C05458=1043.146,323.202,382.853,172.338,41.617,158.001
C05459=1043.153,323.449,382.817,172.342,41.620,158.002
C05460=1043.160,323.697,382.782,172.346,41.623,158.003
C05461=1043.167,323.944,382.748,172.350,41.626,158.003
C05462=1043.174,324.192,382.713,172.355,41.629,158.004
C05463=1043.181,324.439,382.679,172.359,41.631,158.005
C05464=1043.189,324.687,382.643,172.364,41.634,158.006
C05465=1043.196,324.934,382.609,172.369,41.637,158.007
C05466=1043.203,325.181,382.574,172.373,41.640,158.008
C05467=1043.210,325.429,382.538,172.377,41.643,158.009
C05468=1043.218,325.677,382.504,172.382,41.645,158.010
C05469=1043.225,325.924,382.468,172.386,41.649,158.011
C05470=1043.232,326.171,382.434,172.390,41.652,158.012
C05471=1043.239,326.419,382.399,172.395,41.654,158.013
C05472=1043.247,326.667,382.365,172.399,41.657,158.014
C05473=1043.254,326.914,382.329,172.403,41.660,158.014
C05474=1043.260,327.161,382.294,172.408,41.663,158.015
C05475=1043.268,327.408,382.260,172.412,41.666,158.016
C05476=1043.275,327.656,382.224,172.416,41.669,158.017
C05477=1043.283,327.903,382.189,172.422,41.672,158.018
C05478=1043.290,328.150,382.154,172.425,41.675,158.019
C05479=1043.297,328.398,382.118,172.431,41.678,158.020
C05480=1043.305,328.645,382.084,172.435,41.681,158.021
C05481=1043.312,328.894,382.048,172.439,41.683,158.022
C05482=1043.319,329.141,382.013,172.444,41.686,158.023
C05483=1043.326,329.388,381.978,172.448,41.689,158.024
C05484=1043.334,329.635,381.942,172.452,41.693,158.025
C05485=1043.341,329.883,381.907,172.457,41.696,158.026
C05486=1043.348,330.130,381.872,172.461,41.699,158.027
C05487=1043.355,330.378,381.836,172.467,41.702,158.028
C05488=1043.362,330.625,381.801,172.471,41.705,158.029
C05489=1043.369,330.872,381.766,172.475,41.708,158.030
C05490=1043.376,331.120,381.729,172.480,41.711,158.031
C05491=1043.382,331.367,381.694,172.484,41.714,158.032
C05492=1043.389,331.614,381.658,172.489,41.717,158.033
C05493=1043.397,331.862,381.622,172.493,41.720,158.034
C05494=1043.404,332.109,381.587,172.498,41.723,158.035
C05495=1043.411,332.357,381.551,172.503,41.726,158.036
C05496=1043.418,332.604,381.515,172.507,41.730,158.037
C05497=1043.425,332.851,381.480,172.512,41.733,158.038
C05498=1043.433,333.099,381.444,172.516,41.736,158.039
C05499=1043.443,333.428,381.396,172.523,41.740,158.040
C05500=1043.452,333.760,381.349,172.528,41.744,158.041
C05501=1043.462,334.090,381.301,172.535,41.749,158.043
C05502=1043.472,334.420,381.253,172.541,41.753,158.044
C05503=1043.479,334.667,381.217,172.546,41.756,158.045
C05504=1043.486,334.915,381.182,172.551,41.759,158.046
C05505=1043.493,335.162,381.146,172.555,41.762,158.047
C05506=1043.501,335.409,381.110,172.560,41.765,158.048
C05507=1043.508,335.656,381.074,172.564,41.768,158.049
C05508=1043.515,335.904,381.038,172.569,41.772,158.050
C05509=1043.522,336.151,381.002,172.574,41.775,158.051
C05510=1043.529,336.399,380.966,172.578,41.778,158.052
C05511=1043.536,336.645,380.930,172.583,41.782,158.053
C05512=1043.543,336.893,380.893,172.588,41.785,158.054
C05513=1043.550,337.140,380.857,172.593,41.788,158.055
C05514=1043.558,337.387,380.821,172.598,41.792,158.057
C05515=1043.565,337.635,380.784,172.602,41.795,158.058
C05516=1043.572,337.882,380.748,172.608,41.798,158.059
C05517=1043.580,338.129,380.712,172.612,41.801,158.060
C05518=1043.588,338.377,380.676,172.617,41.804,158.061
C05519=1043.594,338.624,380.639,172.621,41.808,158.062
C05520=1043.602,338.871,380.603,172.626,41.811,158.063
C05521=1043.609,339.118,380.567,172.631,41.815,158.064
C05522=1043.616,339.366,380.531,172.636,41.818,158.065
C05523=1043.623,339.613,380.494,172.640,41.821,158.066
C05524=1043.631,339.861,380.458,172.645,41.824,158.067
C05525=1043.637,340.108,380.422,172.651,41.828,158.068
C05526=1043.645,340.355,380.385,172.655,41.831,158.069
C05527=1043.653,340.602,380.349,172.660,41.835,158.070
C05528=1043.660,340.849,380.313,172.665,41.838,158.072
C05529=1043.667,341.096,380.276,172.670,41.841,158.073
C05530=1043.675,341.344,380.240,172.675,41.845,158.074
C05531=1043.682,341.591,380.203,172.679,41.848,158.075
C05532=1043.689,341.838,380.166,172.685,41.851,158.076
C05533=1043.697,342.085,380.130,172.689,41.855,158.077
C05534=1043.704,342.333,380.093,172.694,41.858,158.078
C05535=1043.711,342.580,380.056,172.699,41.862,158.079
C05536=1043.718,342.828,380.020,172.704,41.865,158.080
C05537=1043.726,343.074,379.983,172.709,41.869,158.081
C05538=1043.733,343.321,379.946,172.714,41.872,158.082
C05539=1043.741,343.568,379.909,172.719,41.875,158.084
C05540=1043.748,343.816,379.872,172.724,41.879,158.085
C05541=1043.755,344.063,379.835,172.729,41.883,158.086
C05542=1043.762,344.310,379.799,172.734,41.886,158.087
C05543=1043.769,344.557,379.761,172.739,41.889,158.088
C05544=1043.777,344.804,379.725,172.744,41.893,158.089
C05545=1043.784,345.052,379.688,172.749,41.896,158.090
C05546=1043.792,345.299,379.652,172.754,41.900,158.092
C05547=1043.799,345.546,379.614,172.759,41.904,158.093
C05548=1043.806,345.793,379.576,172.764,41.907,158.094
C05549=1043.814,346.041,379.540,172.769,41.911,158.095
C05550=1043.821,346.288,379.503,172.775,41.914,158.096
C05551=1043.828,346.534,379.466,172.779,41.918,158.097
C05552=1043.836,346.781,379.429,172.784,41.921,158.099
C05553=1043.843,347.029,379.392,172.790,41.925,158.100
C05554=1043.850,347.276,379.354,172.795,41.929,158.101
C05555=1043.860,347.603,379.305,172.802,41.933,158.102
C05556=1043.870,347.929,379.256,172.809,41.938,158.104
C05557=1043.880,348.256,379.207,172.815,41.943,158.106
C05558=1043.890,348.583,379.158,172.821,41.947,158.107
C05559=1043.897,348.830,379.120,172.827,41.952,158.108
C05560=1043.905,349.077,379.083,172.832,41.955,158.109
C05561=1043.912,349.324,379.046,172.838,41.959,158.111
C05562=1043.920,349.571,379.008,172.843,41.962,158.112
C05563=1043.927,349.818,378.971,172.847,41.966,158.113
C05564=1043.935,350.065,378.934,172.853,41.969,158.114
C05565=1043.942,350.312,378.896,172.858,41.973,158.115
C05566=1043.949,350.559,378.859,172.864,41.977,158.117
C05567=1043.957,350.807,378.821,172.869,41.980,158.118
C05568=1043.965,351.054,378.783,172.874,41.985,158.119
C05569=1043.972,351.301,378.745,172.879,41.988,158.120
C05570=1043.979,351.548,378.708,172.884,41.992,158.121
C05571=1043.987,351.795,378.671,172.890,41.996,158.123
C05572=1043.994,352.042,378.633,172.895,41.999,158.124
C05573=1044.002,352.288,378.595,172.901,42.003,158.125
C05574=1044.009,352.535,378.557,172.905,42.007,158.126
C05575=1044.017,352.783,378.519,172.911,42.011,158.128
C05576=1044.025,353.030,378.481,172.916,42.015,158.129
C05577=1044.032,353.277,378.444,172.922,42.019,158.130
C05578=1044.039,353.523,378.405,172.927,42.022,158.131
C05579=1044.047,353.771,378.368,172.933,42.026,158.133
C05580=1044.055,354.018,378.330,172.938,42.030,158.134
C05581=1044.062,354.265,378.292,172.944,42.034,158.135
C05582=1044.069,354.512,378.254,172.948,42.038,158.136
C05583=1044.077,354.759,378.216,172.954,42.042,158.138
C05584=1044.085,355.006,378.178,172.959,42.046,158.139
C05585=1044.092,355.253,378.140,172.965,42.049,158.140
C05586=1044.100,355.500,378.102,172.970,42.053,158.142
C05587=1044.107,355.747,378.064,172.976,42.057,158.143
C05588=1044.115,355.994,378.025,172.981,42.061,158.144
C05589=1044.122,356.241,377.988,172.987,42.065,158.145
C05590=1044.131,356.487,377.950,172.992,42.069,158.147
C05591=1044.139,356.734,377.912,172.998,42.073,158.148
C05592=1044.145,356.982,377.874,173.003,42.077,158.149
C05593=1044.153,357.228,377.835,173.009,42.081,158.151
C05594=1044.161,357.475,377.797,173.015,42.085,158.152
C05595=1044.169,357.722,377.758,173.020,42.089,158.153
C05596=1044.177,357.970,377.721,173.026,42.093,158.155
C05597=1044.184,358.216,377.682,173.031,42.096,158.156
C05598=1044.192,358.463,377.644,173.037,42.100,158.157
C05599=1044.199,358.710,377.605,173.042,42.105,158.158
C05600=1044.207,358.957,377.567,173.048,42.109,158.160
C05601=1044.215,359.204,377.528,173.054,42.113,158.161
C05602=1044.222,359.451,377.490,173.059,42.117,158.162
C05603=1044.230,359.698,377.451,173.065,42.121,158.164
C05604=1044.238,359.944,377.413,173.070,42.125,158.165
C05605=1044.245,360.191,377.374,173.076,42.129,158.166
C05606=1044.253,360.438,377.335,173.082,42.133,158.168
C05607=1044.261,360.685,377.297,173.087,42.138,158.169
C05608=1044.269,360.932,377.259,173.093,42.142,158.171
C05609=1044.276,361.180,377.219,173.099,42.146,158.172
C05610=1044.284,361.426,377.180,173.104,42.150,158.173
C05611=1044.294,361.758,377.129,173.112,42.155,158.175
C05612=1044.305,362.091,377.077,173.120,42.161,158.177
C05613=1044.315,362.423,377.024,173.128,42.166,158.179
C05614=1044.326,362.755,376.972,173.135,42.172,158.181
C05615=1044.333,363.003,376.932,173.141,42.177,158.182
C05616=1044.341,363.249,376.894,173.147,42.181,158.184
C05617=1044.349,363.496,376.854,173.153,42.185,158.185
C05618=1044.356,363.743,376.816,173.159,42.189,158.186
C05619=1044.365,363.989,376.777,173.165,42.193,158.188
C05620=1044.372,364.237,376.738,173.170,42.198,158.189
C05621=1044.380,364.483,376.699,173.176,42.202,158.191
C05622=1044.387,364.730,376.659,173.182,42.206,158.192
C05623=1044.396,364.977,376.620,173.187,42.211,158.193
C05624=1044.403,365.223,376.580,173.194,42.215,158.195
C05625=1044.411,365.470,376.542,173.200,42.219,158.196
C05626=1044.419,365.717,376.502,173.206,42.224,158.198
C05627=1044.425,365.964,376.463,173.212,42.228,158.199
C05628=1044.434,366.210,376.424,173.217,42.232,158.201
C05629=1044.442,366.457,376.384,173.223,42.237,158.202
C05630=1044.450,366.703,376.345,173.230,42.241,158.204
C05631=1044.457,366.951,376.306,173.235,42.245,158.205
C05632=1044.465,367.197,376.266,173.241,42.250,158.207
C05633=1044.473,367.444,376.226,173.247,42.255,158.208
C05634=1044.482,367.691,376.187,173.254,42.258,158.209
C05635=1044.489,367.937,376.148,173.260,42.263,158.211
C05636=1044.497,368.184,376.108,173.265,42.268,158.212
C05637=1044.505,368.431,376.069,173.271,42.272,158.214
C05638=1044.513,368.678,376.030,173.278,42.277,158.215
C05639=1044.521,368.925,375.990,173.284,42.281,158.217
C05640=1044.529,369.171,375.950,173.289,42.285,158.218
C05641=1044.537,369.418,375.911,173.296,42.290,158.220
C05642=1044.545,369.665,375.871,173.302,42.294,158.221
C05643=1044.552,369.911,375.832,173.308,42.299,158.223
C05644=1044.560,370.158,375.792,173.314,42.303,158.224
C05645=1044.569,370.404,375.752,173.321,42.308,158.226
C05646=1044.577,370.651,375.712,173.327,42.312,158.227
C05647=1044.585,370.897,375.672,173.333,42.317,158.229
C05648=1044.593,371.144,375.633,173.339,42.321,158.230
C05649=1044.601,371.391,375.593,173.345,42.327,158.232
C05650=1044.609,371.637,375.552,173.352,42.331,158.234
C05651=1044.616,371.884,375.512,173.358,42.336,158.235
C05652=1044.624,372.131,375.472,173.364,42.340,158.237
C05653=1044.633,372.377,375.432,173.371,42.345,158.238
C05654=1044.641,372.624,375.392,173.377,42.350,158.240
C05655=1044.649,372.870,375.352,173.383,42.354,158.241
C05656=1044.656,373.117,375.312,173.389,42.359,158.243
C05657=1044.664,373.364,375.271,173.395,42.364,158.245
C05658=1044.672,373.611,375.231,173.402,42.368,158.246
C05659=1044.680,373.857,375.190,173.408,42.373,158.248
C05660=1044.688,374.104,375.151,173.414,42.378,158.249
C05661=1044.697,374.350,375.111,173.421,42.383,158.251
C05662=1044.705,374.597,375.070,173.427,42.388,158.253
C05663=1044.713,374.844,375.030,173.434,42.393,158.254
C05664=1044.721,375.090,374.989,173.440,42.397,158.256
C05665=1044.729,375.336,374.948,173.447,42.402,158.258
C05666=1044.737,375.583,374.908,173.453,42.407,158.259
C05667=1044.748,375.935,374.850,173.462,42.414,158.261
C05668=1044.760,376.287,374.793,173.472,42.421,158.264
C05669=1044.772,376.639,374.734,173.481,42.427,158.266
C05670=1044.783,376.991,374.676,173.490,42.434,158.268
C05671=1044.792,377.237,374.636,173.497,42.439,158.270
C05672=1044.800,377.483,374.596,173.504,42.444,158.272
C05673=1044.809,377.730,374.555,173.510,42.449,158.273
C05674=1044.817,377.976,374.514,173.517,42.454,158.275
C05675=1044.825,378.223,374.473,173.524,42.459,158.277
C05676=1044.833,378.470,374.432,173.530,42.464,158.278
C05677=1044.841,378.716,374.392,173.537,42.469,158.280
C05678=1044.849,378.962,374.351,173.543,42.474,158.282
C05679=1044.858,379.209,374.310,173.550,42.479,158.283
C05680=1044.866,379.455,374.270,173.557,42.484,158.285
C05681=1044.874,379.702,374.229,173.563,42.489,158.287
C05682=1044.882,379.948,374.187,173.570,42.494,158.289
C05683=1044.890,380.195,374.146,173.576,42.499,158.290
C05684=1044.898,380.441,374.105,173.584,42.504,158.292
C05685=1044.907,380.687,374.064,173.591,42.509,158.294
C05686=1044.915,380.934,374.022,173.597,42.514,158.296
C05687=1044.924,381.180,373.981,173.604,42.519,158.297
C05688=1044.932,381.427,373.940,173.610,42.525,158.299
C05689=1044.940,381.674,373.899,173.617,42.530,158.301
C05690=1044.948,381.920,373.857,173.624,42.535,158.303
C05691=1044.956,382.165,373.816,173.632,42.540,158.304
C05692=1044.965,382.412,373.775,173.638,42.545,158.306
C05693=1044.973,382.658,373.733,173.645,42.550,158.308
C05694=1044.981,382.905,373.692,173.652,42.556,158.310
C05695=1044.990,383.151,373.650,173.658,42.561,158.311
C05696=1044.998,383.397,373.609,173.666,42.566,158.313
C05697=1045.006,383.644,373.567,173.673,42.571,158.315
C05698=1045.014,383.890,373.526,173.680,42.577,158.317
C05699=1045.023,384.136,373.484,173.686,42.582,158.319
C05700=1045.032,384.382,373.443,173.694,42.587,158.320
C05701=1045.040,384.629,373.401,173.701,42.593,158.322
C05702=1045.049,384.876,373.359,173.708,42.598,158.324
C05703=1045.057,385.121,373.318,173.714,42.603,158.326
C05704=1045.065,385.368,373.276,173.722,42.609,158.328
C05705=1045.074,385.615,373.234,173.729,42.614,158.330
C05706=1045.082,385.860,373.193,173.736,42.620,158.332
C05707=1045.091,386.107,373.151,173.743,42.625,158.333
C05708=1045.099,386.353,373.109,173.751,42.630,158.335
C05709=1045.108,386.600,373.067,173.757,42.636,158.337
C05710=1045.117,386.845,373.026,173.764,42.641,158.339
C05711=1045.125,387.092,372.983,173.772,42.647,158.341
C05712=1045.134,387.338,372.942,173.779,42.652,158.343
C05713=1045.143,387.585,372.900,173.786,42.658,158.345
C05714=1045.151,387.831,372.857,173.794,42.663,158.347
C05715=1045.160,388.077,372.815,173.801,42.669,158.348
C05716=1045.169,388.323,372.774,173.808,42.674,158.350
C05717=1045.177,388.569,372.731,173.816,42.679,158.352
C05718=1045.186,388.815,372.689,173.823,42.685,158.354
C05719=1045.194,389.062,372.647,173.831,42.691,158.356
C05720=1045.203,389.308,372.605,173.838,42.696,158.358
C05721=1045.212,389.554,372.562,173.844,42.702,158.360
C05722=1045.220,389.801,372.520,173.852,42.708,158.362
C05723=1045.231,390.093,372.469,173.861,42.714,158.364
C05724=1045.241,390.386,372.419,173.870,42.721,158.367
C05725=1045.251,390.679,372.368,173.879,42.728,158.369
C05726=1045.261,390.971,372.318,173.888,42.735,158.371
C05727=1045.270,391.218,372.275,173.895,42.740,158.373
C05728=1045.279,391.464,372.233,173.903,42.746,158.375
C05729=1045.287,391.710,372.190,173.910,42.752,158.377
C05730=1045.296,391.956,372.147,173.917,42.758,158.379
C05731=1045.305,392.202,372.105,173.925,42.763,158.381
C05732=1045.313,392.448,372.062,173.934,42.769,158.383
C05733=1045.322,392.694,372.019,173.941,42.775,158.385
C05734=1045.331,392.941,371.976,173.949,42.781,158.387
C05735=1045.340,393.187,371.933,173.956,42.787,158.389
C05736=1045.349,393.433,371.890,173.964,42.793,158.391
C05737=1045.357,393.679,371.847,173.971,42.799,158.394
C05738=1045.366,393.925,371.804,173.979,42.805,158.396
C05739=1045.375,394.171,371.762,173.987,42.811,158.398
C05740=1045.383,394.417,371.719,173.994,42.817,158.400
C05741=1045.392,394.663,371.675,174.003,42.822,158.402
C05742=1045.401,394.910,371.632,174.010,42.828,158.404
C05743=1045.411,395.155,371.589,174.018,42.834,158.406
C05744=1045.419,395.401,371.546,174.026,42.840,158.408
C05745=1045.428,395.647,371.503,174.033,42.846,158.410
C05746=1045.437,395.893,371.460,174.042,42.852,158.412
C05747=1045.445,396.139,371.416,174.050,42.858,158.414
C05748=1045.454,396.385,371.373,174.057,42.864,158.417
C05749=1045.463,396.631,371.329,174.065,42.871,158.419
C05750=1045.472,396.877,371.286,174.074,42.877,158.421
C05751=1045.481,397.123,371.242,174.081,42.883,158.423
C05752=1045.490,397.369,371.199,174.089,42.889,158.425
C05753=1045.499,397.615,371.155,174.097,42.895,158.427
C05754=1045.508,397.862,371.111,174.106,42.901,158.430
C05755=1045.516,398.107,371.068,174.114,42.908,158.432
C05756=1045.526,398.352,371.025,174.121,42.914,158.434
C05757=1045.535,398.599,370.981,174.130,42.920,158.436
C05758=1045.544,398.844,370.937,174.138,42.926,158.438
C05759=1045.553,399.090,370.893,174.145,42.932,158.440
C05760=1045.562,399.336,370.850,174.154,42.939,158.443
C05761=1045.571,399.583,370.806,174.162,42.945,158.445
C05762=1045.580,399.828,370.762,174.171,42.952,158.447
C05763=1045.589,400.074,370.718,174.179,42.957,158.449
C05764=1045.599,400.320,370.674,174.187,42.964,158.452
C05765=1045.608,400.566,370.630,174.195,42.970,158.454
C05766=1045.616,400.812,370.586,174.203,42.977,158.456
C05767=1045.625,401.058,370.542,174.212,42.983,158.458
C05768=1045.635,401.304,370.498,174.220,42.989,158.461
C05769=1045.644,401.550,370.454,174.229,42.996,158.463
C05770=1045.653,401.795,370.410,174.237,43.003,158.465
C05771=1045.662,402.041,370.366,174.246,43.009,158.468
C05772=1045.671,402.287,370.321,174.254,43.015,158.470
C05773=1045.681,402.533,370.276,174.263,43.022,158.472
C05774=1045.689,402.779,370.233,174.271,43.029,158.475
C05775=1045.702,403.117,370.171,174.283,43.037,158.478
C05776=1045.715,403.456,370.110,174.294,43.047,158.481
C05777=1045.728,403.793,370.049,174.306,43.056,158.484
C05778=1045.740,404.131,369.988,174.318,43.065,158.488
C05779=1045.756,404.536,369.914,174.332,43.076,158.492
C05780=1045.770,404.941,369.840,174.346,43.087,158.496
C05781=1045.786,405.345,369.767,174.360,43.098,158.500
C05782=1045.802,405.749,369.693,174.376,43.109,158.504
C05783=1045.810,405.995,369.647,174.384,43.116,158.506
C05784=1045.820,406.241,369.603,174.393,43.123,158.508
C05785=1045.829,406.487,369.558,174.402,43.130,158.511
C05786=1045.839,406.732,369.513,174.410,43.137,158.513
C05787=1045.848,406.978,369.468,174.419,43.144,158.516
C05788=1045.857,407.223,369.423,174.428,43.150,158.518
C05789=1045.866,407.469,369.377,174.438,43.157,158.521
C05790=1045.876,407.715,369.333,174.447,43.164,158.523
C05791=1045.885,407.961,369.287,174.455,43.172,158.526
C05792=1045.895,408.206,369.242,174.464,43.178,158.528
C05793=1045.904,408.452,369.198,174.473,43.185,158.531
C05794=1045.914,408.697,369.151,174.483,43.192,158.533
C05795=1045.924,408.943,369.106,174.492,43.199,158.536
C05796=1045.933,409.189,369.061,174.500,43.207,158.539
C05797=1045.943,409.434,369.016,174.509,43.213,158.541
C05798=1045.952,409.680,368.970,174.519,43.221,158.544
C05799=1045.962,409.926,368.925,174.528,43.228,158.546
C05800=1045.971,410.172,368.879,174.537,43.235,158.549
C05801=1045.981,410.417,368.834,174.547,43.242,158.552
C05802=1045.991,410.663,368.788,174.556,43.249,158.554
C05803=1046.001,410.908,368.742,174.565,43.256,158.557
C05804=1046.010,411.155,368.697,174.575,43.263,158.559
C05805=1046.020,411.400,368.650,174.584,43.271,158.562
C05806=1046.030,411.645,368.605,174.594,43.278,158.565
C05807=1046.039,411.891,368.559,174.603,43.285,158.567
C05808=1046.050,412.137,368.513,174.613,43.292,158.570
C05809=1046.059,412.383,368.468,174.622,43.300,158.573
C05810=1046.070,412.628,368.422,174.631,43.307,158.575
C05811=1046.079,412.873,368.376,174.641,43.315,158.578
C05812=1046.089,413.119,368.329,174.650,43.322,158.581
C05813=1046.098,413.364,368.283,174.661,43.329,158.583
C05814=1046.108,413.610,368.237,174.671,43.337,158.586
C05815=1046.117,413.856,368.190,174.680,43.344,158.589
C05816=1046.128,414.101,368.145,174.690,43.352,158.592
C05817=1046.137,414.346,368.098,174.699,43.359,158.594
C05818=1046.147,414.592,368.052,174.709,43.367,158.597
C05819=1046.157,414.838,368.005,174.719,43.375,158.600
C05820=1046.166,415.083,367.959,174.729,43.382,158.603
C05821=1046.176,415.329,367.912,174.739,43.389,158.606
C05822=1046.186,415.575,367.866,174.748,43.397,158.608
C05823=1046.197,415.819,367.819,174.758,43.405,158.611
C05824=1046.206,416.065,367.773,174.769,43.412,158.614
C05825=1046.217,416.310,367.726,174.778,43.420,158.617
C05826=1046.227,416.556,367.679,174.788,43.428,158.620
C05827=1046.236,416.801,367.632,174.799,43.436,158.623
C05828=1046.246,417.046,367.586,174.809,43.443,158.626
C05829=1046.256,417.292,367.539,174.818,43.451,158.628
C05830=1046.266,417.538,367.492,174.829,43.459,158.631
C05831=1046.277,417.783,367.445,174.839,43.466,158.634
C05832=1046.287,418.028,367.398,174.850,43.474,158.637
C05833=1046.297,418.274,367.352,174.859,43.482,158.640
C05834=1046.307,418.519,367.305,174.870,43.490,158.643
C05835=1046.324,418.930,367.225,174.888,43.503,158.648
C05836=1046.341,419.343,367.145,174.904,43.517,158.653
C05837=1046.358,419.754,367.066,174.922,43.530,158.658
C05838=1046.375,420.166,366.986,174.940,43.544,158.663
C05839=1046.386,420.412,366.939,174.951,43.552,158.666
C05840=1046.396,420.657,366.892,174.962,43.560,158.669
C05841=1046.405,420.902,366.844,174.972,43.568,158.672
C05842=1046.416,421.147,366.796,174.983,43.576,158.676
C05843=1046.426,421.392,366.749,174.994,43.584,158.679
C05844=1046.436,421.638,366.702,175.004,43.593,158.682
C05845=1046.447,421.883,366.653,175.015,43.601,158.685
C05846=1046.457,422.128,366.606,175.026,43.609,158.688
C05847=1046.467,422.373,366.558,175.036,43.617,158.691
C05848=1046.477,422.619,366.510,175.047,43.625,158.694
C05849=1046.489,422.864,366.462,175.058,43.634,158.697
C05850=1046.499,423.109,366.414,175.069,43.642,158.700
C05851=1046.509,423.354,366.367,175.080,43.651,158.704
C05852=1046.520,423.599,366.319,175.090,43.659,158.707
C05853=1046.530,423.844,366.270,175.102,43.667,158.710
C05854=1046.541,424.090,366.222,175.113,43.676,158.713
C05855=1046.552,424.334,366.174,175.124,43.684,158.717
C05856=1046.562,424.580,366.126,175.135,43.693,158.720
C05857=1046.572,424.825,366.078,175.147,43.701,158.723
C05858=1046.583,425.071,366.030,175.158,43.710,158.726
C05859=1046.594,425.315,365.981,175.169,43.718,158.730
C05860=1046.604,425.560,365.932,175.181,43.727,158.733
C05861=1046.615,425.805,365.884,175.192,43.735,158.736
C05862=1046.625,426.051,365.835,175.203,43.744,158.739
C05863=1046.636,426.296,365.787,175.215,43.753,158.743
C05864=1046.647,426.540,365.738,175.226,43.761,158.746
C05865=1046.658,426.786,365.689,175.238,43.770,158.750
C05866=1046.668,427.030,365.641,175.249,43.779,158.753
C05867=1046.679,427.275,365.592,175.261,43.788,158.756
C05868=1046.690,427.520,365.543,175.273,43.797,158.760
C05869=1046.701,427.766,365.494,175.284,43.805,158.763
C05870=1046.711,428.010,365.445,175.296,43.814,158.767
C05871=1046.723,428.255,365.396,175.308,43.823,158.770
C05872=1046.733,428.500,365.347,175.319,43.832,158.773
C05873=1046.744,428.745,365.298,175.332,43.841,158.777
C05874=1046.755,428.990,365.249,175.343,43.850,158.780
C05875=1046.766,429.235,365.199,175.355,43.859,158.784
C05876=1046.777,429.479,365.150,175.368,43.868,158.787
C05877=1046.787,429.724,365.101,175.379,43.877,158.791
C05878=1046.798,429.969,365.051,175.391,43.886,158.794
C05879=1046.809,430.214,365.002,175.404,43.895,158.798
C05880=1046.820,430.459,364.953,175.416,43.904,158.802
C05881=1046.831,430.704,364.903,175.427,43.914,158.805
C05882=1046.842,430.948,364.853,175.440,43.922,158.809
C05883=1046.853,431.193,364.804,175.452,43.932,158.812
C05884=1046.864,431.438,364.754,175.465,43.941,158.816
C05885=1046.875,431.683,364.704,175.477,43.951,158.820
C05886=1046.886,431.928,364.655,175.490,43.960,158.823
C05887=1046.897,432.172,364.604,175.502,43.969,158.827
C05888=1046.908,432.418,364.554,175.514,43.979,158.831
C05889=1046.920,432.662,364.505,175.527,43.988,158.835
C05890=1046.931,432.907,364.455,175.539,43.997,158.838
C05891=1046.941,433.124,364.410,175.551,44.006,158.841
C05892=1046.951,433.342,364.366,175.562,44.014,158.845
C05893=1046.961,433.559,364.321,175.573,44.022,158.848
C05894=1046.971,433.776,364.276,175.585,44.030,158.851
C05895=1046.981,433.993,364.233,175.596,44.039,158.855
C05896=1046.991,434.210,364.188,175.608,44.048,158.858
C05897=1047.001,434.428,364.143,175.618,44.056,158.862
C05898=1047.012,434.644,364.098,175.630,44.065,158.865
C05899=1047.023,434.889,364.048,175.643,44.074,158.869
C05900=1047.034,435.134,363.997,175.656,44.084,158.873
C05901=1047.045,435.378,363.947,175.669,44.094,158.877
C05902=1047.058,435.623,363.897,175.683,44.103,158.880
C05903=1047.069,435.868,363.846,175.696,44.113,158.884
C05904=1047.080,436.112,363.795,175.709,44.123,158.888
C05905=1047.092,436.357,363.744,175.722,44.133,158.892
C05906=1047.103,436.601,363.693,175.736,44.142,158.896
C05907=1047.115,436.846,363.643,175.749,44.152,158.900
C05908=1047.126,437.090,363.592,175.762,44.162,158.904
C05909=1047.138,437.335,363.541,175.776,44.172,158.908
C05910=1047.150,437.580,363.489,175.789,44.182,158.912
C05911=1047.161,437.824,363.438,175.803,44.192,158.916
C05912=1047.173,438.068,363.387,175.817,44.202,158.920
C05913=1047.184,438.313,363.336,175.831,44.212,158.925
C05914=1047.196,438.558,363.285,175.844,44.223,158.929
C05915=1047.208,438.802,363.234,175.858,44.233,158.933
C05916=1047.219,439.046,363.182,175.872,44.243,158.937
C05917=1047.232,439.290,363.130,175.886,44.253,158.941
C05918=1047.243,439.534,363.079,175.900,44.263,158.945
C05919=1047.255,439.779,363.028,175.914,44.273,158.949
C05920=1047.267,440.023,362.976,175.928,44.283,158.954
C05921=1047.279,440.268,362.925,175.941,44.294,158.958
C05922=1047.291,440.512,362.873,175.956,44.304,158.962
C05923=1047.303,440.756,362.821,175.970,44.314,158.966
C05924=1047.315,441.000,362.769,175.985,44.325,158.971
C05925=1047.327,441.245,362.718,175.998,44.335,158.975
C05926=1047.339,441.490,362.665,176.013,44.346,158.979
C05927=1047.351,441.733,362.612,176.028,44.356,158.984
C05928=1047.363,441.978,362.561,176.042,44.367,158.988
C05929=1047.376,442.222,362.509,176.057,44.378,158.992
C05930=1047.388,442.466,362.457,176.071,44.388,158.997
C05931=1047.399,442.710,362.404,176.086,44.399,159.001
C05932=1047.412,442.955,362.352,176.101,44.409,159.006
C05933=1047.424,443.198,362.300,176.116,44.420,159.010
C05934=1047.436,443.442,362.247,176.130,44.431,159.014
C05935=1047.448,443.687,362.194,176.145,44.442,159.019
C05936=1047.461,443.931,362.142,176.160,44.452,159.023
C05937=1047.473,444.174,362.089,176.175,44.463,159.028
C05938=1047.486,444.419,362.037,176.191,44.474,159.033
C05939=1047.497,444.663,361.984,176.206,44.485,159.037
C05940=1047.510,444.907,361.931,176.221,44.496,159.042
C05941=1047.523,445.151,361.879,176.236,44.507,159.046
C05942=1047.536,445.395,361.826,176.252,44.518,159.051
C05943=1047.548,445.638,361.773,176.267,44.529,159.056
C05944=1047.561,445.880,361.721,176.282,44.540,159.060
C05945=1047.575,446.124,361.668,176.298,44.550,159.065
C05946=1047.589,446.368,361.617,176.314,44.561,159.069
C05947=1047.604,446.612,361.566,176.330,44.571,159.074
C05948=1047.620,446.855,361.516,176.345,44.582,159.078
C05949=1047.636,447.099,361.466,176.361,44.592,159.083
C05950=1047.654,447.343,361.417,176.377,44.602,159.087
C05951=1047.680,447.713,361.343,176.401,44.617,159.094
C05952=1047.709,448.082,361.271,176.425,44.632,159.101
C05953=1047.739,448.452,361.200,176.450,44.646,159.107
C05954=1047.771,448.823,361.129,176.474,44.660,159.114
C05955=1047.793,449.067,361.083,176.491,44.669,159.118
C05956=1047.815,449.312,361.038,176.508,44.678,159.122
C05957=1047.838,449.558,360.994,176.525,44.687,159.126
C05958=1047.862,449.802,360.949,176.541,44.696,159.131
C05959=1047.886,450.048,360.906,176.558,44.704,159.135
C05960=1047.911,450.294,360.862,176.575,44.713,159.139
C05961=1047.937,450.539,360.820,176.592,44.721,159.143
C05962=1047.964,450.783,360.778,176.609,44.729,159.147
C05963=1047.654,450.817,360.473,176.610,44.817,159.173
C05964=1047.628,450.571,360.515,176.593,44.809,159.169
C05965=1047.602,450.325,360.557,176.575,44.801,159.165
C05966=1047.576,450.080,360.601,176.559,44.792,159.161
C05967=1047.552,449.835,360.644,176.542,44.784,159.157
C05968=1047.528,449.590,360.688,176.525,44.775,159.152
C05969=1047.505,449.344,360.733,176.508,44.767,159.148
C05970=1047.482,449.100,360.778,176.492,44.757,159.144
C05971=1047.460,448.854,360.824,176.475,44.748,159.140
C05972=1047.430,448.502,360.890,176.451,44.735,159.133
C05973=1047.401,448.149,360.958,176.428,44.722,159.127
C05974=1047.373,447.797,361.027,176.404,44.708,159.121
C05975=1047.346,447.445,361.096,176.381,44.694,159.114
C05976=1047.330,447.201,361.146,176.365,44.684,159.110
C05977=1047.312,446.957,361.196,176.349,44.674,159.105
C05978=1047.296,446.713,361.246,176.333,44.664,159.101
C05979=1047.280,446.469,361.296,176.317,44.654,159.096
C05980=1047.266,446.226,361.347,176.302,44.643,159.092
C05981=1047.252,445.982,361.399,176.287,44.632,159.087
C05982=1047.239,445.739,361.451,176.270,44.622,159.083
C05983=1047.225,445.496,361.503,176.255,44.611,159.078
C05984=1047.213,445.252,361.556,176.240,44.600,159.073
C05985=1047.201,445.008,361.610,176.224,44.589,159.069
C05986=1047.188,444.764,361.662,176.209,44.578,159.064
C05987=1047.175,444.520,361.715,176.194,44.567,159.060
C05988=1047.163,444.276,361.767,176.179,44.557,159.055
C05989=1047.150,444.032,361.820,176.164,44.546,159.051
C05990=1047.139,443.788,361.873,176.148,44.535,159.046
C05991=1047.126,443.544,361.926,176.133,44.524,159.041
C05992=1047.114,443.300,361.978,176.118,44.514,159.037
C05993=1047.101,443.056,362.030,176.103,44.503,159.033
C05994=1047.089,442.811,362.083,176.089,44.493,159.028
C05995=1047.077,442.567,362.135,176.074,44.482,159.024
C05996=1047.065,442.323,362.187,176.059,44.471,159.019
C05997=1047.053,442.079,362.239,176.044,44.461,159.015
C05998=1047.041,441.835,362.291,176.030,44.450,159.010
C05999=1047.028,441.590,362.345,176.015,44.440,159.006
C06000=1047.017,441.346,362.396,176.000,44.429,159.002
C06001=1047.004,441.102,362.448,175.986,44.419,158.997
C06002=1046.993,440.858,362.499,175.972,44.409,158.993
C06003=1046.980,440.614,362.552,175.958,44.398,158.989
C06004=1046.968,440.369,362.603,175.943,44.388,158.985
C06005=1046.956,440.125,362.655,175.929,44.378,158.980
C06006=1046.944,439.881,362.707,175.915,44.368,158.976
C06007=1046.933,439.636,362.758,175.901,44.357,158.972
C06008=1046.920,439.392,362.810,175.887,44.347,158.968
C06009=1046.908,439.148,362.861,175.873,44.337,158.964
C06010=1046.897,438.903,362.913,175.859,44.327,158.959
C06011=1046.885,438.659,362.965,175.845,44.317,158.955
C06012=1046.874,438.414,363.016,175.831,44.307,158.951
C06013=1046.862,438.170,363.067,175.818,44.297,158.947
C06014=1046.850,437.926,363.119,175.804,44.287,158.943
C06015=1046.839,437.681,363.169,175.790,44.277,158.939
C06016=1046.826,437.436,363.220,175.776,44.267,158.935
C06017=1046.815,437.193,363.271,175.763,44.257,158.931
C06018=1046.803,436.948,363.323,175.749,44.247,158.927
C06019=1046.791,436.703,363.373,175.736,44.238,158.923
C06020=1046.780,436.459,363.424,175.723,44.228,158.919
C06021=1046.769,436.214,363.475,175.709,44.218,158.915
C06022=1046.757,435.970,363.526,175.696,44.208,158.911
C06023=1046.746,435.725,363.577,175.683,44.198,158.907
C06024=1046.734,435.480,363.628,175.669,44.189,158.903
C06025=1046.722,435.236,363.677,175.656,44.180,158.899
C06026=1046.711,434.991,363.729,175.643,44.170,158.895
C06027=1046.700,434.747,363.779,175.630,44.160,158.892
C06028=1046.689,434.528,363.824,175.618,44.152,158.888
C06029=1046.679,434.311,363.869,175.607,44.143,158.885
C06030=1046.669,434.092,363.914,175.595,44.135,158.881
C06031=1046.658,433.874,363.958,175.584,44.127,158.878
C06032=1046.649,433.656,364.003,175.572,44.118,158.875
C06033=1046.638,433.438,364.048,175.560,44.109,158.871
C06034=1046.628,433.219,364.093,175.549,44.101,158.868
C06035=1046.618,433.001,364.137,175.539,44.093,158.865
C06036=1046.607,432.757,364.188,175.526,44.083,158.861
C06037=1046.595,432.512,364.237,175.513,44.074,158.857
C06038=1046.585,432.267,364.287,175.501,44.065,158.853
C06039=1046.574,432.022,364.337,175.488,44.055,158.850
C06040=1046.562,431.777,364.387,175.475,44.046,158.846
C06041=1046.551,431.532,364.436,175.463,44.037,158.842
C06042=1046.540,431.288,364.487,175.450,44.028,158.839
C06043=1046.529,431.043,364.536,175.438,44.019,158.835
C06044=1046.518,430.798,364.585,175.425,44.009,158.831
C06045=1046.507,430.554,364.636,175.414,44.000,158.828
C06046=1046.496,430.309,364.685,175.401,43.991,158.824
C06047=1046.485,430.064,364.734,175.389,43.982,158.821
C06048=1046.474,429.819,364.784,175.376,43.973,158.817
C06049=1046.463,429.574,364.833,175.365,43.964,158.814
C06050=1046.452,429.329,364.882,175.353,43.955,158.810
C06051=1046.442,429.085,364.932,175.340,43.946,158.807
C06052=1046.431,428.840,364.981,175.329,43.937,158.803
C06053=1046.420,428.595,365.030,175.317,43.928,158.800
C06054=1046.409,428.350,365.080,175.304,43.920,158.796
C06055=1046.398,428.105,365.128,175.293,43.911,158.793
C06056=1046.387,427.860,365.178,175.281,43.902,158.789
C06057=1046.376,427.615,365.227,175.270,43.893,158.786
C06058=1046.366,427.370,365.275,175.257,43.885,158.782
C06059=1046.355,427.125,365.324,175.246,43.876,158.779
C06060=1046.344,426.880,365.373,175.234,43.867,158.776
C06061=1046.333,426.635,365.422,175.223,43.859,158.772
C06062=1046.323,426.390,365.470,175.211,43.850,158.769
C06063=1046.312,426.144,365.519,175.200,43.841,158.766
C06064=1046.301,425.900,365.568,175.189,43.833,158.762
C06065=1046.290,425.655,365.616,175.177,43.824,158.759
C06066=1046.280,425.409,365.665,175.166,43.815,158.755
C06067=1046.270,425.165,365.713,175.154,43.807,158.752
C06068=1046.259,424.920,365.762,175.143,43.798,158.749
C06069=1046.248,424.675,365.810,175.132,43.790,158.746
C06070=1046.238,424.429,365.858,175.120,43.781,158.742
C06071=1046.227,424.184,365.906,175.109,43.773,158.739
C06072=1046.216,423.939,365.954,175.098,43.765,158.736
C06073=1046.206,423.694,366.003,175.087,43.756,158.733
C06074=1046.195,423.449,366.051,175.076,43.748,158.730
C06075=1046.185,423.204,366.099,175.064,43.740,158.726
C06076=1046.174,422.959,366.146,175.053,43.732,158.723
C06077=1046.163,422.713,366.194,175.042,43.723,158.720
C06078=1046.154,422.468,366.243,175.032,43.715,158.717
C06079=1046.143,422.223,366.290,175.021,43.707,158.714
C06080=1046.132,421.978,366.339,175.010,43.698,158.711
C06081=1046.122,421.732,366.386,174.999,43.690,158.707
C06082=1046.112,421.488,366.434,174.988,43.682,158.704
C06083=1046.101,421.242,366.481,174.977,43.674,158.701
C06084=1046.091,420.996,366.529,174.966,43.666,158.698
C06085=1046.081,420.751,366.577,174.956,43.658,158.695
C06086=1046.071,420.506,366.624,174.945,43.650,158.692
C06087=1046.060,420.261,366.671,174.934,43.642,158.689
C06088=1046.044,419.847,366.752,174.917,43.628,158.684
C06089=1046.026,419.434,366.831,174.899,43.615,158.679
C06090=1046.009,419.020,366.912,174.881,43.602,158.674
C06091=1045.992,418.606,366.991,174.864,43.588,158.669
C06092=1045.982,418.361,367.038,174.854,43.580,158.666
C06093=1045.972,418.115,367.085,174.843,43.573,158.663
C06094=1045.962,417.870,367.132,174.833,43.565,158.660
C06095=1045.952,417.624,367.179,174.823,43.557,158.657
C06096=1045.941,417.379,367.226,174.813,43.549,158.654
C06097=1045.931,417.134,367.273,174.802,43.541,158.651
C06098=1045.921,416.888,367.319,174.792,43.534,158.648
C06099=1045.910,416.643,367.366,174.782,43.526,158.645
C06100=1045.901,416.397,367.413,174.772,43.518,158.643
C06101=1045.891,416.152,367.460,174.762,43.511,158.640
C06102=1045.881,415.906,367.506,174.752,43.504,158.637
C06103=1045.871,415.660,367.553,174.742,43.496,158.634
C06104=1045.861,415.415,367.600,174.732,43.488,158.631
C06105=1045.851,415.170,367.646,174.722,43.480,158.628
C06106=1045.841,414.924,367.692,174.712,43.473,158.626
C06107=1045.831,414.679,367.739,174.702,43.466,158.623
C06108=1045.822,414.434,367.785,174.692,43.458,158.620
C06109=1045.812,414.188,367.832,174.683,43.451,158.617
C06110=1045.802,413.942,367.878,174.673,43.443,158.614
C06111=1045.792,413.697,367.924,174.663,43.436,158.612
C06112=1045.782,413.451,367.970,174.653,43.429,158.609
C06113=1045.773,413.206,368.017,174.643,43.421,158.606
C06114=1045.763,412.960,368.063,174.634,43.414,158.604
C06115=1045.753,412.715,368.109,174.625,43.406,158.601
C06116=1045.744,412.469,368.156,174.615,43.399,158.598
C06117=1045.734,412.224,368.201,174.606,43.392,158.595
C06118=1045.724,411.978,368.248,174.596,43.385,158.593
C06119=1045.713,411.732,368.293,174.587,43.377,158.590
C06120=1045.704,411.487,368.339,174.576,43.370,158.587
C06121=1045.694,411.241,368.384,174.567,43.363,158.585
C06122=1045.685,410.995,368.430,174.557,43.356,158.582
C06123=1045.674,410.750,368.476,174.548,43.348,158.579
C06124=1045.665,410.504,368.522,174.539,43.342,158.577
C06125=1045.655,410.259,368.567,174.529,43.334,158.574
C06126=1045.646,410.013,368.613,174.520,43.327,158.572
C06127=1045.636,409.767,368.658,174.511,43.320,158.569
C06128=1045.626,409.522,368.704,174.502,43.313,158.566
C06129=1045.617,409.276,368.749,174.493,43.306,158.564
C06130=1045.607,409.030,368.795,174.484,43.299,158.561
C06131=1045.597,408.785,368.840,174.474,43.292,158.559
C06132=1045.588,408.539,368.886,174.465,43.285,158.556
C06133=1045.578,408.293,368.930,174.456,43.278,158.554
C06134=1045.569,408.048,368.976,174.447,43.271,158.551
C06135=1045.559,407.801,369.021,174.437,43.265,158.549
C06136=1045.550,407.556,369.066,174.429,43.258,158.546
C06137=1045.540,407.310,369.111,174.420,43.250,158.544
C06138=1045.531,407.064,369.157,174.411,43.244,158.541
C06139=1045.522,406.819,369.202,174.401,43.237,158.539
C06140=1045.512,406.573,369.246,174.393,43.230,158.536
C06141=1045.503,406.327,369.292,174.384,43.223,158.534
C06142=1045.493,406.082,369.337,174.375,43.216,158.531
C06143=1045.484,405.836,369.382,174.366,43.210,158.529
C06144=1045.469,405.430,369.456,174.352,43.199,158.525
C06145=1045.454,405.023,369.530,174.338,43.188,158.521
C06146=1045.438,404.617,369.604,174.322,43.176,158.517
C06147=1045.423,404.211,369.678,174.308,43.166,158.513
C06148=1045.414,403.965,369.723,174.299,43.159,158.510
C06149=1045.405,403.719,369.768,174.291,43.152,158.508
C06150=1045.395,403.473,369.812,174.282,43.146,158.506
C06151=1045.385,403.227,369.857,174.274,43.139,158.503
C06152=1045.377,402.981,369.901,174.265,43.132,158.501
C06153=1045.368,402.735,369.945,174.256,43.126,158.499
C06154=1045.358,402.490,369.990,174.248,43.120,158.496
C06155=1045.349,402.244,370.034,174.239,43.113,158.494
C06156=1045.340,401.997,370.079,174.231,43.106,158.492
C06157=1045.331,401.752,370.122,174.222,43.100,158.489
C06158=1045.322,401.506,370.167,174.214,43.094,158.487
C06159=1045.312,401.260,370.211,174.206,43.088,158.485
C06160=1045.303,401.015,370.255,174.198,43.081,158.482
C06161=1045.294,400.769,370.299,174.189,43.075,158.480
C06162=1045.285,400.523,370.343,174.181,43.068,158.478
C06163=1045.276,400.277,370.387,174.172,43.062,158.476
C06164=1045.266,400.031,370.431,174.164,43.056,158.473
C06165=1045.257,399.784,370.475,174.156,43.050,158.471
C06166=1045.248,399.539,370.518,174.148,43.043,158.469
C06167=1045.239,399.293,370.562,174.140,43.037,158.467
C06168=1045.230,399.047,370.606,174.131,43.031,158.464
C06169=1045.221,398.801,370.650,174.123,43.025,158.462
C06170=1045.212,398.555,370.693,174.115,43.018,158.460
C06171=1045.203,398.309,370.737,174.106,43.012,158.458
C06172=1045.194,398.064,370.781,174.099,43.006,158.456
C06173=1045.185,397.817,370.825,174.091,43.000,158.453
C06174=1045.176,397.571,370.868,174.082,42.994,158.451
C06175=1045.167,397.326,370.912,174.074,42.988,158.449
C06176=1045.158,397.079,370.955,174.067,42.981,158.447
C06177=1045.150,396.834,370.999,174.058,42.976,158.445
C06178=1045.141,396.588,371.042,174.050,42.969,158.443
C06179=1045.132,396.342,371.086,174.042,42.963,158.441
C06180=1045.123,396.095,371.129,174.035,42.957,158.438
C06181=1045.114,395.850,371.173,174.026,42.952,158.436
C06182=1045.106,395.604,371.216,174.018,42.945,158.434
C06183=1045.096,395.358,371.259,174.011,42.939,158.432
C06184=1045.087,395.111,371.302,174.003,42.933,158.430
C06185=1045.079,394.866,371.346,173.994,42.927,158.428
C06186=1045.070,394.619,371.389,173.987,42.921,158.426
C06187=1045.061,394.373,371.432,173.979,42.915,158.424
C06188=1045.052,394.128,371.475,173.972,42.909,158.422
C06189=1045.043,393.881,371.518,173.964,42.904,158.419
C06190=1045.035,393.635,371.561,173.956,42.898,158.418
C06191=1045.026,393.389,371.604,173.948,42.892,158.415
C06192=1045.016,393.143,371.646,173.940,42.886,158.413
C06193=1045.008,392.897,371.689,173.933,42.880,158.411
C06194=1044.999,392.651,371.732,173.925,42.874,158.409
C06195=1044.990,392.405,371.775,173.918,42.869,158.407
C06196=1044.980,392.106,371.827,173.909,42.862,158.405
C06197=1044.970,391.806,371.879,173.899,42.855,158.402
C06198=1044.959,391.507,371.932,173.889,42.848,158.400
C06199=1044.948,391.207,371.983,173.880,42.841,158.397
C06200=1044.936,390.874,372.041,173.870,42.834,158.395
C06201=1044.924,390.539,372.099,173.860,42.825,158.392
C06202=1044.913,390.205,372.156,173.850,42.818,158.389
C06203=1044.901,389.872,372.214,173.840,42.810,158.387
C06204=1044.893,389.626,372.256,173.832,42.805,158.385
C06205=1044.884,389.379,372.298,173.825,42.799,158.383
C06206=1044.876,389.133,372.341,173.818,42.794,158.381
C06207=1044.867,388.887,372.383,173.810,42.788,158.379
C06208=1044.858,388.641,372.426,173.803,42.782,158.377
C06209=1044.849,388.394,372.467,173.795,42.777,158.375
C06210=1044.841,388.148,372.510,173.788,42.772,158.373
C06211=1044.832,387.902,372.552,173.781,42.766,158.371
C06212=1044.823,387.656,372.594,173.773,42.761,158.369
C06213=1044.815,387.410,372.636,173.766,42.755,158.367
C06214=1044.806,387.163,372.677,173.758,42.750,158.366
C06215=1044.797,386.917,372.719,173.752,42.744,158.364
C06216=1044.789,386.670,372.761,173.745,42.739,158.362
C06217=1044.780,386.424,372.803,173.738,42.734,158.360
C06218=1044.772,386.178,372.845,173.730,42.728,158.358
C06219=1044.763,385.932,372.888,173.723,42.723,158.356
C06220=1044.755,385.685,372.929,173.715,42.717,158.354
C06221=1044.746,385.439,372.970,173.708,42.713,158.353
C06222=1044.738,385.193,373.012,173.701,42.707,158.351
C06223=1044.729,384.946,373.054,173.695,42.701,158.349
C06224=1044.720,384.700,373.096,173.687,42.697,158.347
C06225=1044.712,384.454,373.137,173.680,42.691,158.345
C06226=1044.704,384.208,373.179,173.673,42.686,158.344
C06227=1044.696,383.962,373.221,173.666,42.681,158.342
C06228=1044.687,383.715,373.262,173.660,42.676,158.340
C06229=1044.678,383.469,373.303,173.652,42.670,158.338
C06230=1044.670,383.223,373.345,173.645,42.665,158.336
C06231=1044.662,382.976,373.386,173.638,42.660,158.334
C06232=1044.653,382.730,373.428,173.632,42.655,158.333
C06233=1044.645,382.483,373.470,173.624,42.649,158.331
C06234=1044.637,382.237,373.511,173.617,42.644,158.329
C06235=1044.628,381.991,373.552,173.611,42.639,158.327
C06236=1044.620,381.744,373.593,173.604,42.634,158.326
C06237=1044.612,381.498,373.635,173.597,42.629,158.324
C06238=1044.604,381.251,373.676,173.589,42.624,158.322
C06239=1044.595,381.005,373.718,173.583,42.619,158.320
C06240=1044.587,380.759,373.758,173.576,42.614,158.319
C06241=1044.579,380.512,373.801,173.569,42.608,158.317
C06242=1044.571,380.266,373.841,173.563,42.603,158.315
C06243=1044.563,380.020,373.882,173.556,42.598,158.313
C06244=1044.554,379.773,373.924,173.550,42.593,158.312
C06245=1044.547,379.527,373.965,173.542,42.588,158.310
C06246=1044.539,379.280,374.005,173.535,42.583,158.308
C06247=1044.530,379.033,374.046,173.529,42.578,158.307
C06248=1044.522,378.788,374.088,173.522,42.573,158.305
C06249=1044.514,378.541,374.128,173.516,42.568,158.303
C06250=1044.505,378.294,374.169,173.509,42.564,158.302
C06251=1044.497,378.048,374.210,173.502,42.559,158.300
C06252=1044.488,377.802,374.250,173.496,42.554,158.298
C06253=1044.480,377.555,374.291,173.489,42.549,158.296
C06254=1044.472,377.309,374.332,173.483,42.544,158.295
C06255=1044.463,377.063,374.372,173.476,42.539,158.293
C06256=1044.452,376.708,374.431,173.467,42.532,158.291
C06257=1044.440,376.354,374.489,173.457,42.525,158.288
C06258=1044.428,376.000,374.547,173.448,42.518,158.286
C06259=1044.417,375.647,374.605,173.438,42.512,158.284
C06260=1044.408,375.400,374.646,173.432,42.507,158.282
C06261=1044.400,375.153,374.686,173.425,42.502,158.281
C06262=1044.392,374.907,374.727,173.419,42.497,158.279
C06263=1044.384,374.660,374.766,173.412,42.493,158.277
C06264=1044.376,374.414,374.807,173.406,42.488,158.276
C06265=1044.368,374.167,374.847,173.399,42.483,158.274
C06266=1044.360,373.921,374.888,173.393,42.478,158.272
C06267=1044.351,373.674,374.929,173.386,42.474,158.271
C06268=1044.344,373.427,374.968,173.380,42.469,158.269
C06269=1044.336,373.181,375.009,173.373,42.464,158.268
C06270=1044.328,372.934,375.049,173.368,42.460,158.266
C06271=1044.319,372.688,375.089,173.362,42.455,158.265
C06272=1044.311,372.441,375.129,173.355,42.451,158.263
C06273=1044.303,372.195,375.170,173.349,42.446,158.261
C06274=1044.296,371.948,375.210,173.342,42.441,158.260
C06275=1044.288,371.701,375.249,173.336,42.437,158.258
C06276=1044.280,371.455,375.290,173.330,42.432,158.257
C06277=1044.272,371.208,375.330,173.323,42.428,158.255
C06278=1044.264,370.961,375.369,173.317,42.423,158.254
C06279=1044.256,370.714,375.409,173.311,42.419,158.252
C06280=1044.248,370.468,375.450,173.305,42.414,158.251
C06281=1044.240,370.222,375.489,173.299,42.410,158.249
C06282=1044.232,369.975,375.529,173.293,42.405,158.248
C06283=1044.224,369.729,375.568,173.286,42.401,158.246
C06284=1044.216,369.482,375.608,173.280,42.396,158.245
C06285=1044.208,369.235,375.647,173.274,42.391,158.243
C06286=1044.200,368.988,375.687,173.267,42.387,158.241
C06287=1044.192,368.741,375.727,173.262,42.383,158.240
C06288=1044.184,368.495,375.766,173.256,42.378,158.239
C06289=1044.176,368.248,375.806,173.249,42.374,158.237
C06290=1044.168,368.001,375.846,173.243,42.369,158.236
C06291=1044.161,367.755,375.885,173.238,42.365,158.234
C06292=1044.153,367.508,375.924,173.232,42.361,158.233
C06293=1044.145,367.261,375.964,173.225,42.356,158.231
C06294=1044.136,367.014,376.003,173.219,42.352,158.230
C06295=1044.129,366.767,376.043,173.213,42.348,158.228
C06296=1044.121,366.521,376.082,173.208,42.343,158.227
C06297=1044.113,366.274,376.121,173.201,42.339,158.225
C06298=1044.105,366.027,376.161,173.195,42.335,158.224
C06299=1044.097,365.780,376.200,173.189,42.331,158.223
C06300=1044.090,365.534,376.239,173.184,42.326,158.221
C06301=1044.082,365.287,376.279,173.178,42.321,158.219
C06302=1044.073,365.040,376.318,173.171,42.318,158.218
C06303=1044.067,364.794,376.357,173.165,42.314,158.217
C06304=1044.058,364.547,376.396,173.160,42.309,158.215
C06305=1044.051,364.299,376.435,173.154,42.305,158.214
C06306=1044.043,364.054,376.474,173.148,42.300,158.212
C06307=1044.035,363.806,376.513,173.143,42.296,158.211
C06308=1044.027,363.559,376.553,173.136,42.292,158.210
C06309=1044.020,363.313,376.592,173.130,42.288,158.208
C06310=1044.012,363.066,376.631,173.124,42.284,158.207
C06311=1044.005,362.819,376.670,173.119,42.279,158.205
C06312=1043.994,362.484,376.722,173.111,42.273,158.203
C06313=1043.984,362.150,376.775,173.103,42.268,158.202
C06314=1043.973,361.816,376.827,173.095,42.262,158.200
C06315=1043.962,361.481,376.880,173.088,42.257,158.198
C06316=1043.954,361.235,376.919,173.082,42.253,158.197
C06317=1043.947,360.988,376.958,173.076,42.249,158.195
C06318=1043.939,360.741,376.996,173.071,42.245,158.194
C06319=1043.931,360.494,377.035,173.064,42.241,158.192
C06320=1043.924,360.247,377.073,173.059,42.237,158.191
C06321=1043.916,360.000,377.112,173.053,42.233,158.190
C06322=1043.909,359.753,377.151,173.047,42.229,158.188
C06323=1043.901,359.506,377.189,173.042,42.225,158.187
C06324=1043.893,359.260,377.228,173.036,42.221,158.186
C06325=1043.885,359.012,377.266,173.030,42.217,158.184
C06326=1043.877,358.766,377.304,173.025,42.212,158.183
C06327=1043.870,358.519,377.343,173.019,42.208,158.182
C06328=1043.862,358.272,377.382,173.014,42.204,158.180
C06329=1043.855,358.025,377.420,173.008,42.200,158.179
C06330=1043.847,357.778,377.459,173.003,42.197,158.178
C06331=1043.839,357.532,377.497,172.997,42.193,158.177
C06332=1043.832,357.285,377.535,172.991,42.189,158.175
C06333=1043.824,357.037,377.573,172.986,42.185,158.174
C06334=1043.816,356.791,377.611,172.980,42.181,158.172
C06335=1043.809,356.544,377.650,172.975,42.177,158.171
C06336=1043.801,356.296,377.688,172.969,42.173,158.170
C06337=1043.793,356.050,377.726,172.963,42.169,158.169
C06338=1043.786,355.803,377.764,172.958,42.165,158.167
C06339=1043.778,355.556,377.802,172.952,42.161,158.166
C06340=1043.770,355.309,377.840,172.947,42.158,158.165
C06341=1043.763,355.062,377.878,172.941,42.154,158.164
C06342=1043.755,354.815,377.916,172.936,42.150,158.162
C06343=1043.748,354.568,377.954,172.930,42.146,158.161
C06344=1043.740,354.321,377.992,172.926,42.142,158.160
C06345=1043.733,354.074,378.030,172.920,42.139,158.159
C06346=1043.725,353.827,378.068,172.915,42.134,158.157
C06347=1043.717,353.580,378.106,172.909,42.131,158.156
C06348=1043.710,353.333,378.144,172.904,42.127,158.155
C06349=1043.703,353.086,378.182,172.898,42.123,158.154
C06350=1043.695,352.839,378.219,172.893,42.120,158.152
C06351=1043.687,352.592,378.258,172.887,42.116,158.151
C06352=1043.680,352.344,378.295,172.882,42.112,158.150
C06353=1043.672,352.098,378.332,172.877,42.108,158.149
C06354=1043.665,351.851,378.370,172.872,42.105,158.147
C06355=1043.657,351.604,378.408,172.867,42.101,158.146
C06356=1043.650,351.357,378.445,172.861,42.097,158.145
C06357=1043.643,351.110,378.483,172.856,42.093,158.144
C06358=1043.635,350.862,378.521,172.850,42.090,158.142
C06359=1043.627,350.615,378.559,172.846,42.086,158.141
C06360=1043.620,350.368,378.597,172.840,42.082,158.140
C06361=1043.613,350.121,378.634,172.835,42.079,158.139
C06362=1043.605,349.874,378.671,172.829,42.075,158.138
C06363=1043.598,349.627,378.709,172.824,42.072,158.136
C06364=1043.590,349.380,378.746,172.819,42.068,158.135
C06365=1043.582,349.133,378.783,172.814,42.065,158.134
C06366=1043.575,348.886,378.821,172.809,42.060,158.133
C06367=1043.568,348.639,378.858,172.803,42.057,158.132
C06368=1043.558,348.310,378.907,172.796,42.052,158.130
C06369=1043.548,347.982,378.958,172.790,42.048,158.129
C06370=1043.538,347.653,379.006,172.783,42.043,158.127
C06371=1043.528,347.325,379.056,172.776,42.038,158.125
C06372=1043.521,347.077,379.093,172.771,42.035,158.124
C06373=1043.513,346.830,379.131,172.766,42.031,158.123
C06374=1043.506,346.583,379.167,172.761,42.027,158.122
C06375=1043.499,346.336,379.205,172.755,42.024,158.121
C06376=1043.491,346.089,379.242,172.750,42.020,158.120
C06377=1043.483,345.842,379.279,172.746,42.017,158.118
C06378=1043.476,345.594,379.316,172.740,42.013,158.117
C06379=1043.468,345.347,379.353,172.735,42.010,158.116
C06380=1043.462,345.101,379.390,172.730,42.007,158.115
C06381=1043.455,344.853,379.427,172.725,42.003,158.114
C06382=1043.447,344.606,379.464,172.720,42.000,158.113
C06383=1043.440,344.358,379.501,172.715,41.996,158.112
C06384=1043.432,344.112,379.537,172.710,41.993,158.111
C06385=1043.425,343.864,379.574,172.705,41.989,158.109
C06386=1043.417,343.617,379.611,172.700,41.986,158.108
C06387=1043.411,343.370,379.648,172.695,41.982,158.107
C06388=1043.403,343.123,379.685,172.690,41.979,158.106
C06389=1043.396,342.875,379.721,172.685,41.976,158.105
C06390=1043.388,342.628,379.759,172.680,41.972,158.104
C06391=1043.381,342.381,379.795,172.675,41.968,158.103
C06392=1043.374,342.134,379.832,172.671,41.965,158.102
C06393=1043.366,341.887,379.868,172.665,41.962,158.100
C06394=1043.359,341.639,379.905,172.660,41.959,158.099
C06395=1043.352,341.392,379.942,172.656,41.955,158.098
C06396=1043.344,341.146,379.978,172.650,41.952,158.097
C06397=1043.337,340.898,380.014,172.645,41.949,158.096
C06398=1043.330,340.650,380.051,172.641,41.945,158.095
C06399=1043.322,340.403,380.087,172.636,41.942,158.094
C06400=1043.315,340.156,380.123,172.630,41.938,158.093
C06401=1043.308,339.909,380.161,172.626,41.935,158.092
C06402=1043.300,339.662,380.197,172.621,41.932,158.091
C06403=1043.293,339.414,380.233,172.617,41.929,158.090
C06404=1043.286,339.167,380.270,172.611,41.926,158.089
C06405=1043.279,338.920,380.306,172.607,41.922,158.088
C06406=1043.271,338.672,380.342,172.602,41.919,158.087
C06407=1043.264,338.425,380.378,172.597,41.916,158.085
C06408=1043.257,338.178,380.415,172.592,41.912,158.084
C06409=1043.250,337.931,380.451,172.587,41.909,158.083
C06410=1043.242,337.684,380.487,172.583,41.906,158.082
C06411=1043.235,337.436,380.524,172.578,41.903,158.081
C06412=1043.228,337.189,380.559,172.573,41.900,158.080
C06413=1043.220,336.942,380.596,172.568,41.896,158.079
C06414=1043.213,336.695,380.631,172.564,41.893,158.078
C06415=1043.206,336.447,380.668,172.559,41.890,158.077
C06416=1043.199,336.200,380.705,172.554,41.886,158.076
C06417=1043.192,335.953,380.740,172.549,41.883,158.075
C06418=1043.184,335.705,380.776,172.545,41.880,158.074
C06419=1043.178,335.458,380.812,172.540,41.877,158.073
C06420=1043.170,335.210,380.849,172.536,41.874,158.072
C06421=1043.163,334.964,380.884,172.530,41.871,158.071
C06422=1043.156,334.715,380.920,172.526,41.867,158.070
C06423=1043.149,334.469,380.956,172.521,41.864,158.069
C06424=1043.139,334.137,381.004,172.515,41.860,158.067
C06425=1043.129,333.804,381.052,172.509,41.856,158.066
C06426=1043.119,333.472,381.100,172.502,41.852,158.065
C06427=1043.110,333.139,381.148,172.496,41.848,158.063
C06428=1043.102,332.892,381.184,172.492,41.845,158.062
C06429=1043.095,332.645,381.220,172.487,41.842,158.061
C06430=1043.088,332.398,381.255,172.482,41.838,158.060
C06431=1043.080,332.150,381.291,172.478,41.835,158.059
C06432=1043.074,331.903,381.326,172.473,41.832,158.058
C06433=1043.066,331.655,381.362,172.469,41.830,158.058
C06434=1043.059,331.408,381.397,172.464,41.827,158.057
C06435=1043.052,331.161,381.433,172.460,41.824,158.056
C06436=1043.045,330.913,381.469,172.454,41.821,158.055
C06437=1043.038,330.666,381.504,172.450,41.818,158.054
C06438=1043.030,330.418,381.540,172.446,41.814,158.053
C06439=1043.024,330.171,381.575,172.441,41.811,158.052
C06440=1043.017,329.924,381.610,172.437,41.808,158.051
C06441=1043.009,329.676,381.647,172.432,41.805,158.050
C06442=1043.002,329.429,381.682,172.427,41.802,158.049
C06443=1042.996,329.182,381.717,172.423,41.799,158.048
C06444=1042.988,328.933,381.752,172.418,41.797,158.047
C06445=1042.981,328.687,381.788,172.414,41.793,158.046
C06446=1042.974,328.440,381.823,172.409,41.790,158.045
C06447=1042.966,328.192,381.858,172.405,41.787,158.044
C06448=1042.959,327.945,381.893,172.401,41.785,158.043
C06449=1042.952,327.697,381.928,172.396,41.782,158.042
C06450=1042.945,327.449,381.963,172.392,41.779,158.041
C06451=1042.937,327.202,381.998,172.387,41.776,158.040
C06452=1042.930,326.955,382.033,172.383,41.773,158.039
C06453=1042.922,326.707,382.068,172.379,41.771,158.038
C06454=1042.916,326.460,382.103,172.373,41.768,158.037
C06455=1042.909,326.212,382.138,172.369,41.764,158.036
C06456=1042.901,325.965,382.173,172.365,41.762,158.036
C06457=1042.894,325.717,382.208,172.360,41.759,158.035
C06458=1042.886,325.470,382.243,172.356,41.756,158.034
C06459=1042.880,325.223,382.278,172.352,41.753,158.033
C06460=1042.873,324.975,382.313,172.347,41.751,158.032
C06461=1042.865,324.727,382.347,172.343,41.748,158.031
C06462=1042.858,324.480,382.382,172.339,41.745,158.030
C06463=1042.851,324.233,382.417,172.334,41.742,158.029
C06464=1042.844,323.985,382.452,172.330,41.739,158.028
C06465=1042.836,323.738,382.487,172.326,41.736,158.027
C06466=1042.830,323.491,382.522,172.321,41.734,158.026
C06467=1042.822,323.242,382.556,172.317,41.731,158.025
C06468=1042.815,322.995,382.591,172.313,41.728,158.025
C06469=1042.808,322.748,382.626,172.309,41.725,158.024
C06470=1042.801,322.501,382.661,172.304,41.723,158.023
C06471=1042.794,322.253,382.695,172.299,41.720,158.022
C06472=1042.787,322.006,382.730,172.295,41.717,158.021
C06473=1042.780,321.758,382.765,172.291,41.714,158.020
C06474=1042.773,321.511,382.799,172.286,41.711,158.019
C06475=1042.766,321.263,382.834,172.282,41.709,158.018
C06476=1042.759,321.016,382.868,172.278,41.706,158.017
C06477=1042.752,320.767,382.903,172.274,41.703,158.017
C06478=1042.744,320.520,382.938,172.269,41.700,158.016
C06479=1042.738,320.272,382.972,172.265,41.698,158.015
C06480=1042.728,319.936,383.019,172.260,41.694,158.014
C06481=1042.719,319.599,383.066,172.253,41.690,158.012
C06482=1042.709,319.261,383.113,172.248,41.686,158.011
C06483=1042.700,318.924,383.160,172.243,41.683,158.010
C06484=1042.693,318.677,383.195,172.238,41.680,158.009
C06485=1042.686,318.429,383.229,172.234,41.677,158.008
C06486=1042.679,318.182,383.264,172.230,41.674,158.007
C06487=1042.672,317.934,383.298,172.226,41.672,158.007
C06488=1042.665,317.686,383.332,172.222,41.669,158.006
C06489=1042.658,317.439,383.367,172.218,41.666,158.005
C06490=1042.652,317.192,383.401,172.213,41.664,158.004
C06491=1042.644,316.945,383.435,172.209,41.661,158.003
C06492=1042.638,316.697,383.470,172.205,41.658,158.002
C06493=1042.631,316.449,383.503,172.201,41.655,158.001
C06494=1042.624,316.202,383.539,172.197,41.653,158.000
C06495=1042.617,315.954,383.572,172.193,41.650,158.000
C06496=1042.610,315.706,383.607,172.189,41.647,157.999
C06497=1042.604,315.459,383.640,172.184,41.645,157.998
C06498=1042.597,315.212,383.675,172.180,41.642,157.997
C06499=1042.590,314.964,383.709,172.176,41.639,157.996
C06500=1042.583,314.716,383.744,172.172,41.637,157.995
C06501=1042.576,314.469,383.777,172.168,41.634,157.994
C06502=1042.570,314.221,383.811,172.164,41.631,157.994
C06503=1042.563,313.974,383.846,172.160,41.629,157.993
C06504=1042.556,313.726,383.880,172.156,41.626,157.992
C06505=1042.549,313.479,383.914,172.152,41.623,157.991
C06506=1042.542,313.232,383.948,172.148,41.621,157.990
C06507=1042.536,312.984,383.982,172.143,41.618,157.989
C06508=1042.529,312.736,384.016,172.139,41.615,157.988
C06509=1042.523,312.489,384.050,172.135,41.613,157.988
C06510=1042.516,312.241,384.084,172.131,41.610,157.987
C06511=1042.508,311.993,384.118,172.127,41.607,157.986
C06512=1042.501,311.746,384.151,172.123,41.605,157.985
C06513=1042.494,311.498,384.185,172.119,41.603,157.985
C06514=1042.487,311.251,384.219,172.116,41.600,157.984
C06515=1042.480,311.003,384.252,172.112,41.598,157.983
C06516=1042.473,310.755,384.285,172.108,41.595,157.982
C06517=1042.465,310.508,384.319,172.103,41.593,157.981
C06518=1042.458,310.260,384.353,172.099,41.590,157.980
C06519=1042.452,310.013,384.386,172.095,41.588,157.980
C06520=1042.445,309.765,384.419,172.091,41.585,157.979
C06521=1042.437,309.517,384.453,172.087,41.583,157.978
C06522=1042.431,309.270,384.487,172.083,41.580,157.977
C06523=1042.424,309.022,384.520,172.079,41.578,157.977
C06524=1042.416,308.774,384.553,172.076,41.576,157.976
C06525=1042.409,308.527,384.587,172.072,41.573,157.975
C06526=1042.403,308.279,384.620,172.068,41.571,157.974
C06527=1042.395,308.032,384.653,172.064,41.568,157.973
C06528=1042.389,307.785,384.687,172.060,41.566,157.973
C06529=1042.382,307.536,384.720,172.056,41.563,157.972
C06530=1042.375,307.289,384.754,172.052,41.561,157.971
C06531=1042.367,307.042,384.787,172.048,41.558,157.970
C06532=1042.360,306.794,384.820,172.044,41.556,157.970
C06533=1042.353,306.546,384.854,172.039,41.554,157.969
C06534=1042.347,306.298,384.886,172.036,41.551,157.968
C06535=1042.340,306.051,384.920,172.032,41.549,157.967
C06536=1042.331,305.718,384.965,172.026,41.546,157.966
C06537=1042.321,305.386,385.009,172.021,41.542,157.965
C06538=1042.312,305.053,385.053,172.016,41.539,157.964
C06539=1042.302,304.721,385.098,172.011,41.536,157.963
C06540=1042.296,304.474,385.131,172.007,41.534,157.962
C06541=1042.289,304.225,385.164,172.003,41.531,157.962
C06542=1042.283,303.978,385.197,171.999,41.529,157.961
C06543=1042.275,303.730,385.231,171.997,41.526,157.960
C06544=1042.269,303.483,385.264,171.993,41.524,157.959
C06545=1042.262,303.235,385.296,171.989,41.521,157.959
C06546=1042.255,302.988,385.330,171.985,41.519,157.958
C06547=1042.248,302.739,385.363,171.981,41.517,157.957
C06548=1042.242,302.492,385.395,171.977,41.514,157.956
C06549=1042.235,302.244,385.429,171.973,41.512,157.956
C06550=1042.228,301.997,385.461,171.969,41.509,157.955
C06551=1042.221,301.749,385.494,171.966,41.507,157.954
C06552=1042.214,301.502,385.528,171.962,41.505,157.953
C06553=1042.208,301.254,385.561,171.958,41.502,157.952
C06554=1042.201,301.006,385.594,171.954,41.500,157.952
C06555=1042.194,300.758,385.626,171.950,41.498,157.951
C06556=1042.187,300.510,385.659,171.946,41.496,157.950
C06557=1042.181,300.263,385.692,171.944,41.493,157.950
C06558=1042.174,300.016,385.725,171.940,41.490,157.949
C06559=1042.167,299.767,385.758,171.936,41.488,157.948
C06560=1042.160,299.520,385.790,171.932,41.486,157.947
C06561=1042.153,299.272,385.824,171.928,41.484,157.947
C06562=1042.147,299.024,385.856,171.924,41.481,157.946
C06563=1042.141,298.776,385.889,171.920,41.479,157.945
C06564=1042.134,298.528,385.922,171.917,41.476,157.944
C06565=1042.127,298.281,385.954,171.914,41.474,157.944
C06566=1042.120,298.033,385.987,171.910,41.472,157.943
C06567=1042.114,297.786,386.020,171.906,41.470,157.942
C06568=1042.107,297.537,386.053,171.902,41.467,157.941
C06569=1042.100,297.290,386.085,171.899,41.465,157.941
C06570=1042.094,297.043,386.118,171.895,41.462,157.940
C06571=1042.087,296.794,386.151,171.892,41.460,157.939
C06572=1042.081,296.547,386.184,171.888,41.458,157.938
C06573=1042.074,296.299,386.216,171.884,41.456,157.938
C06574=1042.067,296.052,386.249,171.880,41.453,157.937
C06575=1042.060,295.803,386.282,171.877,41.451,157.936
C06576=1042.054,295.556,386.314,171.873,41.448,157.936
C06577=1042.047,295.309,386.347,171.870,41.446,157.935
C06578=1042.041,295.060,386.379,171.866,41.444,157.934
C06579=1042.034,294.812,386.411,171.862,41.442,157.933
C06580=1042.027,294.565,386.444,171.858,41.439,157.933
C06581=1042.020,294.318,386.476,171.855,41.437,157.932
C06582=1042.014,294.069,386.508,171.852,41.435,157.931
C06583=1042.007,293.821,386.541,171.848,41.433,157.931
C06584=1042.000,293.574,386.573,171.844,41.431,157.930
C06585=1041.994,293.326,386.605,171.840,41.428,157.929
C06586=1041.987,293.079,386.637,171.837,41.426,157.929
C06587=1041.980,292.830,386.670,171.833,41.424,157.928
C06588=1041.973,292.582,386.701,171.830,41.422,157.927
C06589=1041.966,292.335,386.734,171.826,41.419,157.926
C06590=1041.960,292.087,386.766,171.823,41.417,157.926
C06591=1041.952,291.839,386.798,171.819,41.415,157.925
C06592=1041.944,291.523,386.839,171.815,41.413,157.924
C06593=1041.935,291.207,386.879,171.810,41.409,157.923
C06594=1041.926,290.891,386.921,171.806,41.407,157.923
C06595=1041.918,290.575,386.962,171.801,41.404,157.922
C06596=1041.911,290.327,386.993,171.797,41.402,157.921
C06597=1041.904,290.080,387.026,171.794,41.400,157.920
C06598=1041.898,289.832,387.058,171.791,41.398,157.920
C06599=1041.891,289.584,387.089,171.787,41.396,157.919
C06600=1041.884,289.336,387.122,171.783,41.393,157.918
C06601=1041.877,289.088,387.153,171.780,41.391,157.918
C06602=1041.871,288.841,387.186,171.776,41.389,157.917
C06603=1041.864,288.593,387.217,171.773,41.387,157.916
C06604=1041.857,288.345,387.249,171.769,41.385,157.916
C06605=1041.850,288.098,387.281,171.766,41.383,157.915
C06606=1041.844,287.849,387.313,171.763,41.380,157.914
C06607=1041.838,287.601,387.344,171.759,41.378,157.914
C06608=1041.831,287.354,387.376,171.756,41.376,157.913
C06609=1041.823,287.106,387.408,171.752,41.374,157.912
C06610=1041.817,286.858,387.440,171.748,41.372,157.912
C06611=1041.810,286.610,387.471,171.745,41.370,157.911
C06612=1041.803,286.362,387.502,171.742,41.367,157.910
C06613=1041.796,286.115,387.535,171.738,41.365,157.910
C06614=1041.789,285.867,387.566,171.735,41.363,157.909
C06615=1041.783,285.619,387.597,171.732,41.361,157.908
C06616=1041.777,285.371,387.629,171.728,41.359,157.908
C06617=1041.770,285.123,387.661,171.724,41.357,157.907
C06618=1041.763,284.875,387.692,171.721,41.355,157.906
C06619=1041.756,284.627,387.724,171.718,41.353,157.906
C06620=1041.750,284.379,387.755,171.714,41.351,157.905
C06621=1041.743,284.131,387.787,171.710,41.349,157.904
C06622=1041.736,283.883,387.818,171.708,41.347,157.904
C06623=1041.730,283.635,387.850,171.704,41.345,157.903
C06624=1041.723,283.387,387.881,171.700,41.343,157.902
C06625=1041.716,283.139,387.912,171.698,41.340,157.902
C06626=1041.709,282.891,387.944,171.694,41.338,157.901
C06627=1041.703,282.644,387.975,171.690,41.336,157.900
C06628=1041.696,282.396,388.007,171.687,41.334,157.900
C06629=1041.689,282.148,388.038,171.684,41.332,157.899
C06630=1041.682,281.900,388.070,171.680,41.330,157.899
C06631=1041.676,281.652,388.101,171.677,41.328,157.898
C06632=1041.669,281.404,388.132,171.673,41.326,157.897
C06633=1041.662,281.156,388.164,171.671,41.324,157.897
C06634=1041.656,280.908,388.195,171.667,41.322,157.896
C06635=1041.649,280.660,388.227,171.663,41.320,157.895
C06636=1041.642,280.412,388.258,171.661,41.318,157.895
C06637=1041.635,280.165,388.290,171.657,41.316,157.894
C06638=1041.629,279.916,388.320,171.654,41.314,157.894
C06639=1041.622,279.668,388.352,171.651,41.312,157.893
C06640=1041.615,279.420,388.383,171.647,41.310,157.892
C06641=1041.609,279.173,388.414,171.644,41.308,157.892
C06642=1041.603,278.925,388.446,171.640,41.306,157.891
C06643=1041.595,278.677,388.476,171.638,41.303,157.890
C06644=1041.589,278.429,388.507,171.634,41.301,157.890
C06645=1041.582,278.181,388.539,171.630,41.300,157.889
C06646=1041.576,277.933,388.569,171.628,41.298,157.889
C06647=1041.569,277.685,388.601,171.624,41.296,157.888
C06648=1041.560,277.381,388.638,171.620,41.293,157.887
C06649=1041.552,277.076,388.677,171.616,41.291,157.886
C06650=1041.544,276.773,388.715,171.612,41.288,157.886
C06651=1041.536,276.468,388.752,171.609,41.286,157.885
C06652=1041.529,276.221,388.783,171.605,41.284,157.884
C06653=1041.522,275.972,388.814,171.601,41.282,157.884
C06654=1041.516,275.724,388.845,171.599,41.280,157.883
C06655=1041.509,275.476,388.877,171.595,41.278,157.882
C06656=1041.502,275.229,388.906,171.592,41.276,157.882
C06657=1041.496,274.981,388.938,171.588,41.274,157.881
C06658=1041.489,274.732,388.968,171.586,41.272,157.881
C06659=1041.482,274.484,389.000,171.582,41.270,157.880
C06660=1041.475,274.236,389.030,171.579,41.268,157.879
C06661=1041.469,273.989,389.061,171.576,41.266,157.879
C06662=1041.463,273.740,389.092,171.572,41.265,157.878
C06663=1041.456,273.492,389.122,171.569,41.262,157.878
C06664=1041.449,273.244,389.153,171.566,41.260,157.877
C06665=1041.442,272.996,389.184,171.563,41.258,157.876
C06666=1041.436,272.749,389.215,171.559,41.257,157.876
C06667=1041.429,272.500,389.245,171.557,41.255,157.875
C06668=1041.422,272.252,389.275,171.553,41.252,157.875
C06669=1041.415,272.004,389.307,171.550,41.251,157.874
C06670=1041.409,271.756,389.337,171.547,41.249,157.873
C06671=1041.402,271.508,389.367,171.544,41.247,157.873
C06672=1041.396,271.260,389.399,171.540,41.245,157.872
C06673=1041.388,271.012,389.429,171.538,41.243,157.872
C06674=1041.383,270.764,389.459,171.534,41.241,157.871
C06675=1041.375,270.516,389.489,171.531,41.239,157.870
C06676=1041.369,270.268,389.520,171.528,41.237,157.870
C06677=1041.362,270.020,389.551,171.525,41.235,157.869
C06678=1041.356,269.772,389.581,171.521,41.233,157.869
C06679=1041.349,269.524,389.611,171.519,41.232,157.868
C06680=1041.342,269.275,389.642,171.515,41.229,157.867
C06681=1041.336,269.028,389.672,171.512,41.227,157.867
C06682=1041.329,268.779,389.703,171.509,41.226,157.866
C06683=1041.322,268.532,389.733,171.506,41.224,157.866
C06684=1041.316,268.284,389.764,171.504,41.222,157.865
C06685=1041.309,268.036,389.794,171.500,41.220,157.865
C06686=1041.302,267.787,389.825,171.497,41.218,157.864
C06687=1041.296,267.540,389.854,171.494,41.216,157.863
C06688=1041.289,267.291,389.885,171.491,41.214,157.863
C06689=1041.282,267.043,389.915,171.487,41.213,157.862
C06690=1041.276,266.795,389.945,171.485,41.211,157.862
C06691=1041.269,266.547,389.976,171.481,41.208,157.861
C06692=1041.262,266.299,390.006,171.478,41.207,157.861
C06693=1041.256,266.051,390.036,171.476,41.205,157.860
C06694=1041.249,265.803,390.066,171.472,41.203,157.859
C06695=1041.242,265.554,390.096,171.469,41.201,157.859
C06696=1041.235,265.307,390.126,171.466,41.200,157.858
C06697=1041.229,265.058,390.157,171.463,41.197,157.858
C06698=1041.222,264.811,390.187,171.459,41.195,157.857
C06699=1041.215,264.563,390.217,171.457,41.194,157.857
C06700=1041.209,264.314,390.247,171.454,41.192,157.856
C06701=1041.203,264.066,390.276,171.451,41.190,157.855
C06702=1041.195,263.818,390.307,171.448,41.188,157.855
C06703=1041.190,263.570,390.337,171.444,41.187,157.854
C06704=1041.181,263.270,390.373,171.441,41.184,157.854
C06705=1041.173,262.971,390.409,171.438,41.182,157.853
C06706=1041.165,262.671,390.445,171.434,41.180,157.852
C06707=1041.157,262.371,390.482,171.430,41.177,157.852
C06708=1041.151,262.123,390.512,171.427,41.175,157.851
C06709=1041.144,261.875,390.542,171.424,41.174,157.850
C06710=1041.137,261.628,390.571,171.421,41.172,157.850
C06711=1041.130,261.379,390.601,171.418,41.170,157.849
C06712=1041.123,261.130,390.631,171.415,41.168,157.849
C06713=1041.117,260.883,390.661,171.412,41.167,157.848
C06714=1041.110,260.634,390.690,171.409,41.165,157.848
C06715=1041.103,260.387,390.720,171.406,41.163,157.847
C06716=1041.096,260.138,390.749,171.403,41.161,157.847
C06717=1041.090,259.890,390.779,171.400,41.160,157.846
C06718=1041.082,259.642,390.808,171.397,41.158,157.845
C06719=1041.075,259.394,390.838,171.394,41.156,157.845
C06720=1041.068,259.146,390.868,171.391,41.154,157.844
C06721=1041.062,258.897,390.897,171.388,41.152,157.844
C06722=1041.055,258.650,390.927,171.385,41.151,157.843
C06723=1041.048,258.401,390.956,171.383,41.149,157.843
C06724=1041.042,258.153,390.986,171.379,41.147,157.842
C06725=1041.035,257.905,391.015,171.377,41.146,157.842
C06726=1041.029,257.656,391.045,171.374,41.143,157.841
C06727=1041.021,257.408,391.075,171.370,41.142,157.841
C06728=1041.015,257.160,391.104,171.368,41.140,157.840
C06729=1041.008,256.912,391.134,171.365,41.138,157.840
C06730=1041.002,256.664,391.163,171.362,41.137,157.839
C06731=1040.995,256.415,391.193,171.359,41.134,157.838
C06732=1040.988,256.168,391.221,171.356,41.133,157.838
C06733=1040.981,255.919,391.251,171.353,41.131,157.837
C06734=1040.974,255.671,391.281,171.350,41.129,157.837
C06735=1040.968,255.423,391.310,171.348,41.128,157.836
C06736=1040.961,255.175,391.340,171.344,41.126,157.836
C06737=1040.955,254.927,391.369,171.341,41.124,157.835
C06738=1040.948,254.678,391.398,171.339,41.122,157.835
C06739=1040.941,254.430,391.428,171.335,41.121,157.834
C06740=1040.935,254.182,391.457,171.333,41.119,157.834
C06741=1040.928,253.934,391.486,171.330,41.117,157.833
C06742=1040.921,253.686,391.515,171.327,41.116,157.833
C06743=1040.914,253.437,391.545,171.324,41.113,157.832
C06744=1040.908,253.189,391.574,171.321,41.112,157.832
C06745=1040.901,252.941,391.603,171.319,41.110,157.831
C06746=1040.895,252.692,391.632,171.316,41.108,157.830
C06747=1040.888,252.445,391.662,171.312,41.107,157.830
C06748=1040.882,252.197,391.691,171.310,41.104,157.829
C06749=1040.875,251.948,391.721,171.307,41.103,157.829
C06750=1040.869,251.700,391.750,171.304,41.101,157.828
C06751=1040.862,251.452,391.778,171.301,41.099,157.828
C06752=1040.854,251.204,391.808,171.299,41.097,157.827
C06753=1040.848,250.956,391.837,171.296,41.096,157.827
C06754=1040.842,250.707,391.866,171.293,41.094,157.826
C06755=1040.835,250.459,391.896,171.290,41.092,157.826
C06756=1040.829,250.211,391.925,171.287,41.091,157.825
C06757=1040.823,249.962,391.954,171.285,41.088,157.825
C06758=1040.816,249.714,391.983,171.282,41.087,157.824
C06759=1040.808,249.466,392.012,171.278,41.085,157.823
C06760=1040.801,249.165,392.048,171.276,41.083,157.823
C06761=1040.793,248.864,392.083,171.272,41.080,157.822
C06762=1040.785,248.563,392.118,171.268,41.078,157.822
C06763=1040.777,248.262,392.154,171.265,41.076,157.821
C06764=1040.771,248.014,392.183,171.263,41.075,157.821
C06765=1040.764,247.766,392.212,171.259,41.072,157.820
C06766=1040.758,247.518,392.241,171.257,41.071,157.819
C06767=1040.751,247.269,392.270,171.254,41.069,157.819
C06768=1040.745,247.021,392.299,171.252,41.067,157.818
C06769=1040.738,246.773,392.328,171.249,41.065,157.818
C06770=1040.732,246.525,392.357,171.246,41.064,157.817
C06771=1040.726,246.276,392.386,171.243,41.062,157.817
C06772=1040.719,246.028,392.415,171.240,41.060,157.816
C06773=1040.712,245.779,392.444,171.238,41.059,157.816
C06774=1040.707,245.531,392.473,171.235,41.056,157.815
C06775=1040.700,245.283,392.501,171.232,41.055,157.815
C06776=1040.693,245.035,392.530,171.230,41.053,157.814
C06777=1040.686,244.786,392.559,171.226,41.051,157.814
C06778=1040.679,244.538,392.588,171.224,41.049,157.813
C06779=1040.673,244.290,392.617,171.221,41.048,157.813
C06780=1040.667,244.041,392.645,171.219,41.046,157.812
C06781=1040.660,243.793,392.674,171.216,41.044,157.812
C06782=1040.653,243.545,392.703,171.213,41.042,157.811
C06783=1040.646,243.297,392.732,171.211,41.041,157.811
C06784=1040.640,243.048,392.760,171.207,41.039,157.810
C06785=1040.634,242.800,392.788,171.205,41.037,157.809
C06786=1040.627,242.552,392.817,171.202,41.036,157.809
C06787=1040.621,242.304,392.846,171.200,41.034,157.809
C06788=1040.614,242.055,392.874,171.197,41.032,157.808
C06789=1040.607,241.807,392.904,171.194,41.030,157.807
C06790=1040.600,241.559,392.932,171.192,41.028,157.807
C06791=1040.595,241.310,392.960,171.189,41.027,157.806
C06792=1040.588,241.062,392.989,171.186,41.025,157.806
C06793=1040.581,240.814,393.018,171.183,41.023,157.805
C06794=1040.575,240.566,393.046,171.181,41.022,157.805
C06795=1040.568,240.317,393.075,171.178,41.020,157.804
C06796=1040.561,240.068,393.103,171.176,41.018,157.804
C06797=1040.554,239.821,393.131,171.173,41.017,157.803
C06798=1040.548,239.572,393.159,171.170,41.015,157.803
C06799=1040.541,239.324,393.188,171.168,41.013,157.802
C06800=1040.534,239.076,393.216,171.164,41.011,157.802
C06801=1040.528,238.827,393.245,171.162,41.010,157.801
C06802=1040.521,238.579,393.273,171.159,41.008,157.801
C06803=1040.514,238.330,393.301,171.157,41.007,157.800
C06804=1040.508,238.082,393.329,171.154,41.004,157.800
C06805=1040.501,237.834,393.358,171.152,41.003,157.799
C06806=1040.494,237.585,393.386,171.149,41.001,157.799
C06807=1040.488,237.337,393.415,171.147,41.000,157.798
C06808=1040.481,237.089,393.442,171.144,40.998,157.798
C06809=1040.474,236.841,393.471,171.142,40.996,157.798
C06810=1040.468,236.593,393.499,171.138,40.995,157.797
C06811=1040.462,236.344,393.527,171.135,40.993,157.796
C06812=1040.455,236.096,393.555,171.133,40.991,157.796
C06813=1040.448,235.848,393.583,171.130,40.989,157.795
C06814=1040.441,235.599,393.612,171.128,40.988,157.795
C06815=1040.435,235.350,393.640,171.125,40.986,157.795
C06816=1040.426,235.044,393.675,171.123,40.984,157.794
C06817=1040.418,234.737,393.710,171.119,40.982,157.793
C06818=1040.410,234.430,393.744,171.116,40.980,157.793
C06819=1040.402,234.123,393.779,171.112,40.978,157.792
C06820=1040.395,233.874,393.807,171.110,40.976,157.792
C06821=1040.388,233.627,393.835,171.107,40.974,157.791
C06822=1040.382,233.378,393.863,171.105,40.973,157.791
C06823=1040.376,233.129,393.891,171.102,40.971,157.790
C06824=1040.369,232.881,393.919,171.100,40.969,157.790
C06825=1040.362,232.633,393.947,171.097,40.967,157.789
C06826=1040.356,232.384,393.976,171.095,40.966,157.789
C06827=1040.349,232.136,394.003,171.092,40.964,157.788
C06828=1040.343,231.888,394.031,171.090,40.962,157.788
C06829=1040.336,231.639,394.059,171.087,40.961,157.787
C06830=1040.329,231.391,394.087,171.085,40.959,157.787
C06831=1040.322,231.143,394.115,171.082,40.957,157.786
C06832=1040.316,230.894,394.143,171.079,40.955,157.786
C06833=1040.310,230.646,394.171,171.077,40.954,157.785
C06834=1040.304,230.398,394.198,171.074,40.952,157.785
C06835=1040.297,230.149,394.226,171.072,40.951,157.784
C06836=1040.290,229.901,394.254,171.069,40.949,157.784
C06837=1040.284,229.653,394.282,171.067,40.947,157.783
C06838=1040.277,229.404,394.309,171.064,40.946,157.783
C06839=1040.270,229.156,394.338,171.062,40.943,157.782
C06840=1040.263,228.908,394.366,171.059,40.942,157.782
C06841=1040.257,228.659,394.393,171.057,40.940,157.781
C06842=1040.250,228.411,394.421,171.054,40.939,157.781
C06843=1040.243,228.163,394.449,171.052,40.937,157.780
C06844=1040.237,227.914,394.476,171.049,40.935,157.780
C06845=1040.230,227.666,394.504,171.047,40.934,157.779
C06846=1040.224,227.417,394.531,171.044,40.932,157.779
C06847=1040.217,227.168,394.559,171.042,40.931,157.778
C06848=1040.210,226.920,394.587,171.039,40.929,157.778
C06849=1040.204,226.672,394.614,171.037,40.927,157.777
C06850=1040.197,226.424,394.641,171.034,40.926,157.777
C06851=1040.190,226.175,394.669,171.031,40.924,157.777
C06852=1040.183,225.927,394.697,171.029,40.922,157.776
C06853=1040.177,225.679,394.724,171.026,40.921,157.776
C06854=1040.170,225.430,394.752,171.024,40.919,157.775
C06855=1040.164,225.181,394.779,171.021,40.918,157.775
C06856=1040.157,224.933,394.807,171.019,40.916,157.774
C06857=1040.150,224.684,394.834,171.016,40.914,157.774
C06858=1040.143,224.437,394.861,171.015,40.912,157.773
C06859=1040.137,224.188,394.889,171.012,40.910,157.773
C06860=1040.130,223.939,394.916,171.010,40.909,157.772
C06861=1040.124,223.691,394.944,171.007,40.907,157.772
C06862=1040.117,223.442,394.972,171.005,40.906,157.771
C06863=1040.110,223.194,394.999,171.002,40.904,157.771
C06864=1040.103,222.946,395.026,171.000,40.902,157.770
C06865=1040.097,222.697,395.053,170.997,40.901,157.770
C06866=1040.090,222.449,395.081,170.995,40.899,157.769
C06867=1040.084,222.201,395.109,170.992,40.897,157.769
C06868=1040.077,221.952,395.136,170.990,40.896,157.768
C06869=1040.071,221.703,395.163,170.988,40.894,157.768
C06870=1040.064,221.456,395.190,170.986,40.892,157.768
C06871=1040.057,221.207,395.218,170.983,40.890,157.767
C06872=1040.049,220.892,395.253,170.979,40.889,157.766
C06873=1040.041,220.578,395.287,170.977,40.886,157.766
C06874=1040.032,220.264,395.321,170.974,40.884,157.765
C06875=1040.024,219.949,395.356,170.970,40.882,157.765
C06876=1040.017,219.701,395.382,170.968,40.880,157.764
C06877=1040.011,219.453,395.410,170.965,40.879,157.764
C06878=1040.004,219.204,395.437,170.964,40.877,157.763
C06879=1039.997,218.956,395.464,170.961,40.875,157.763
C06880=1039.991,218.706,395.491,170.959,40.874,157.762
C06881=1039.984,218.459,395.518,170.956,40.872,157.762
C06882=1039.977,218.211,395.546,170.954,40.871,157.761
C06883=1039.971,217.962,395.573,170.951,40.869,157.761
C06884=1039.964,217.713,395.599,170.949,40.867,157.760
C06885=1039.957,217.464,395.627,170.946,40.866,157.760
C06886=1039.950,217.216,395.653,170.945,40.864,157.760
C06887=1039.944,216.968,395.681,170.942,40.862,157.759
C06888=1039.937,216.719,395.707,170.940,40.861,157.759
C06889=1039.930,216.471,395.735,170.937,40.859,157.758
C06890=1039.924,216.222,395.761,170.935,40.857,157.758
C06891=1039.917,215.974,395.789,170.932,40.856,157.757
C06892=1039.910,215.725,395.816,170.931,40.854,157.757
C06893=1039.904,215.478,395.842,170.928,40.852,157.756
C06894=1039.897,215.229,395.869,170.926,40.851,157.756
C06895=1039.890,214.980,395.896,170.923,40.849,157.755
C06896=1039.883,214.731,395.924,170.921,40.848,157.755
C06897=1039.877,214.483,395.950,170.918,40.846,157.754
C06898=1039.871,214.234,395.977,170.917,40.844,157.754
C06899=1039.864,213.986,396.004,170.914,40.843,157.754
C06900=1039.857,213.738,396.030,170.912,40.841,157.753
C06901=1039.851,213.489,396.057,170.909,40.839,157.753
C06902=1039.844,213.241,396.085,170.907,40.838,157.752
C06903=1039.838,212.992,396.111,170.905,40.836,157.752
C06904=1039.831,212.744,396.138,170.902,40.834,157.751
C06905=1039.825,212.496,396.165,170.900,40.832,157.751
C06906=1039.817,212.247,396.191,170.897,40.830,157.750
C06907=1039.811,211.998,396.218,170.895,40.829,157.750
C06908=1039.804,211.751,396.245,170.893,40.827,157.749
C06909=1039.798,211.502,396.272,170.891,40.825,157.749
C06910=1039.791,211.253,396.299,170.888,40.824,157.748
C06911=1039.785,211.004,396.325,170.886,40.822,157.748
C06912=1039.778,210.756,396.352,170.884,40.820,157.747
C06913=1039.770,210.508,396.379,170.882,40.819,157.747
C06914=1039.765,210.259,396.405,170.879,40.817,157.746
C06915=1039.758,210.010,396.432,170.877,40.815,157.746
C06916=1039.751,209.762,396.458,170.874,40.814,157.746
C06917=1039.745,209.513,396.485,170.873,40.812,157.745
C06918=1039.738,209.265,396.511,170.870,40.810,157.745
C06919=1039.732,209.017,396.539,170.868,40.809,157.744
C06920=1039.724,208.768,396.565,170.865,40.807,157.744
C06921=1039.717,208.519,396.592,170.864,40.805,157.743
C06922=1039.711,208.271,396.618,170.861,40.804,157.743
C06923=1039.704,208.022,396.645,170.859,40.802,157.742
C06924=1039.698,207.774,396.671,170.856,40.801,157.742
C06925=1039.691,207.525,396.697,170.855,40.799,157.741
C06926=1039.685,207.277,396.724,170.852,40.797,157.741
C06927=1039.678,207.028,396.750,170.850,40.796,157.741
C06928=1039.670,206.719,396.783,170.847,40.794,157.740
C06929=1039.660,206.411,396.816,170.845,40.792,157.739
C06930=1039.653,206.103,396.848,170.842,40.789,157.739
C06931=1039.644,205.793,396.881,170.840,40.788,157.738
C06932=1039.618,204.742,396.988,170.547,40.684,157.703
C06933=1039.612,204.494,397.013,170.545,40.683,157.702
C06934=1039.606,204.245,397.039,170.541,40.682,157.702
C06935=1039.600,203.996,397.063,170.538,40.681,157.702
C06936=1039.593,203.748,397.088,170.535,40.680,157.701
C06937=1039.587,203.499,397.113,170.532,40.679,157.701
C06938=1039.581,203.251,397.138,170.529,40.678,157.701
C06939=1039.575,203.002,397.164,170.526,40.677,157.700
C06940=1039.569,202.753,397.189,170.522,40.677,157.700
C06941=1039.563,202.504,397.214,170.520,40.675,157.700
C06942=1039.557,202.255,397.239,170.517,40.675,157.700
C06943=1039.551,202.007,397.264,170.513,40.674,157.699
C06944=1039.545,201.759,397.289,170.511,40.673,157.699
C06945=1039.539,201.509,397.314,170.508,40.672,157.699
C06946=1039.533,201.261,397.339,170.504,40.671,157.698
C06947=1039.526,201.012,397.364,170.501,40.670,157.698
C06948=1039.520,200.763,397.388,170.499,40.669,157.698
C06949=1039.514,200.514,397.414,170.495,40.669,157.697
C06950=1039.507,200.267,397.438,170.492,40.668,157.697
C06951=1039.501,200.018,397.463,170.489,40.667,157.697
C06952=1039.494,199.769,397.488,170.486,40.666,157.696
C06953=1039.488,199.520,397.512,170.483,40.666,157.696
C06954=1039.482,199.271,397.538,170.480,40.665,157.696
C06955=1039.476,199.022,397.562,170.478,40.664,157.695
C06956=1039.470,198.774,397.587,170.474,40.664,157.695
C06957=1039.463,198.525,397.611,170.471,40.663,157.695
C06958=1039.457,198.277,397.636,170.468,40.662,157.695
C06959=1039.451,198.028,397.660,170.466,40.662,157.694
C06960=1039.444,197.779,397.685,170.462,40.661,157.694
C06961=1039.439,197.530,397.710,170.459,40.660,157.694
C06962=1039.432,197.282,397.734,170.457,40.659,157.693
C06963=1039.426,197.033,397.759,170.453,40.658,157.693
C06964=1039.419,196.784,397.784,170.450,40.657,157.693
C06965=1039.414,196.536,397.808,170.448,40.657,157.693
C06966=1039.407,196.287,397.833,170.444,40.656,157.692
C06967=1039.401,196.038,397.857,170.441,40.655,157.692
C06968=1039.394,195.789,397.881,170.439,40.655,157.692
C06969=1039.389,195.541,397.906,170.436,40.654,157.691
C06970=1039.383,195.292,397.931,170.432,40.653,157.691
C06971=1039.376,195.044,397.956,170.430,40.653,157.691
C06972=1039.370,194.794,397.980,170.427,40.652,157.690
C06973=1039.364,194.546,398.004,170.423,40.651,157.690
C06974=1039.358,194.297,398.029,170.421,40.650,157.690
C06975=1039.351,194.048,398.053,170.418,40.649,157.690
C06976=1039.346,193.800,398.078,170.415,40.648,157.689
C06977=1039.339,193.551,398.102,170.412,40.648,157.689
C06978=1039.333,193.302,398.127,170.409,40.647,157.689
C06979=1039.327,193.054,398.151,170.406,40.647,157.688
C06980=1039.321,192.805,398.175,170.403,40.646,157.688
C06981=1039.314,192.556,398.200,170.400,40.645,157.688
C06982=1039.309,192.308,398.224,170.397,40.645,157.688
C06983=1039.302,192.059,398.248,170.395,40.644,157.687
C06984=1039.296,191.809,398.273,170.391,40.643,157.687
C06985=1039.290,191.562,398.297,170.389,40.642,157.687
C06986=1039.284,191.312,398.322,170.386,40.641,157.686
C06987=1039.278,191.064,398.345,170.383,40.641,157.686
C06988=1039.272,190.815,398.370,170.380,40.640,157.686
C06989=1039.266,190.566,398.395,170.377,40.640,157.686
C06990=1039.260,190.318,398.419,170.375,40.639,157.685
C06991=1039.254,190.069,398.444,170.372,40.638,157.685
C06992=1039.248,189.820,398.467,170.368,40.637,157.685
C06993=1039.241,189.536,398.495,170.365,40.636,157.684
C06994=1039.234,189.251,398.523,170.361,40.636,157.684
C06995=1039.227,188.968,398.551,170.358,40.635,157.684
C06996=1039.221,188.683,398.578,170.356,40.634,157.684
C06997=1039.214,188.434,398.602,170.353,40.633,157.683
C06998=1039.209,188.185,398.627,170.349,40.633,157.683
C06999=1039.202,187.936,398.651,170.347,40.632,157.683
C07000=1039.197,187.687,398.675,170.344,40.632,157.682
C07001=1039.190,187.439,398.700,170.342,40.631,157.682
C07002=1039.184,187.190,398.724,170.338,40.630,157.682
C07003=1039.178,186.942,398.748,170.336,40.629,157.682
C07004=1039.172,186.693,398.772,170.333,40.628,157.681
C07005=1039.166,186.444,398.796,170.330,40.628,157.681
C07006=1039.160,186.196,398.820,170.327,40.627,157.681
C07007=1039.154,185.946,398.845,170.324,40.627,157.681
C07008=1039.148,185.698,398.868,170.322,40.626,157.680
C07009=1039.142,185.449,398.893,170.318,40.625,157.680
C07010=1039.136,185.201,398.917,170.316,40.624,157.680
C07011=1039.131,184.952,398.941,170.313,40.624,157.680
C07012=1039.124,184.702,398.964,170.311,40.623,157.679
C07013=1039.119,184.454,398.988,170.307,40.623,157.679
C07014=1039.112,184.205,399.012,170.305,40.622,157.679
C07015=1039.107,183.956,399.037,170.302,40.621,157.678
C07016=1039.100,183.707,399.061,170.300,40.620,157.678
C07017=1039.095,183.459,399.085,170.296,40.620,157.678
C07018=1039.089,183.210,399.109,170.294,40.619,157.678
C07019=1039.082,182.961,399.131,170.291,40.619,157.677
C07020=1039.075,182.712,399.155,170.288,40.618,157.677
C07021=1039.069,182.464,399.179,170.286,40.618,157.677
C07022=1039.063,182.215,399.203,170.282,40.618,157.677
C07023=1039.057,181.966,399.226,170.280,40.617,157.676
C07024=1039.050,181.717,399.250,170.277,40.616,157.676
C07025=1039.044,181.469,399.274,170.275,40.616,157.676
C07026=1039.038,181.219,399.297,170.271,40.616,157.676
C07027=1039.032,180.971,399.321,170.268,40.615,157.676
C07028=1039.026,180.721,399.344,170.266,40.614,157.675
C07029=1039.020,180.473,399.368,170.263,40.614,157.675
C07030=1039.012,180.224,399.391,170.261,40.614,157.675
C07031=1039.006,179.975,399.414,170.257,40.613,157.675
C07032=1039.000,179.726,399.438,170.255,40.613,157.675
C07033=1038.994,179.478,399.462,170.252,40.613,157.674
C07034=1038.988,179.229,399.485,170.250,40.611,157.674
C07035=1038.981,178.980,399.509,170.247,40.611,157.674
C07036=1038.976,178.731,399.532,170.244,40.611,157.674
C07037=1038.969,178.482,399.556,170.241,40.610,157.673
C07038=1038.963,178.233,399.579,170.238,40.610,157.673
C07039=1038.956,177.985,399.602,170.236,40.609,157.673
C07040=1038.950,177.736,399.625,170.232,40.609,157.673
C07041=1038.944,177.488,399.649,170.230,40.608,157.672
C07042=1038.938,177.238,399.672,170.227,40.608,157.672
C07043=1038.932,176.990,399.696,170.225,40.608,157.672
C07044=1038.925,176.740,399.719,170.222,40.607,157.672
C07045=1038.919,176.492,399.743,170.220,40.607,157.672
C07046=1038.914,176.243,399.766,170.216,40.606,157.671
C07047=1038.906,175.994,399.789,170.214,40.606,157.671
C07048=1038.901,175.745,399.812,170.211,40.605,157.671
C07049=1038.895,175.497,399.836,170.209,40.605,157.671
C07050=1038.888,175.248,399.859,170.205,40.605,157.671
C07051=1038.883,174.999,399.882,170.203,40.604,157.670
C07052=1038.876,174.750,399.905,170.200,40.604,157.670
C07053=1038.870,174.501,399.929,170.198,40.603,157.670
C07054=1038.864,174.253,399.952,170.195,40.603,157.670
C07055=1038.858,174.004,399.975,170.192,40.602,157.669
C07056=1038.851,173.754,399.998,170.190,40.602,157.669
C07057=1038.845,173.470,400.025,170.187,40.601,157.669
C07058=1038.837,173.185,400.051,170.184,40.600,157.669
C07059=1038.831,172.901,400.078,170.181,40.600,157.669
C07060=1038.823,172.616,400.104,170.177,40.600,157.668
C07061=1038.817,172.367,400.128,170.175,40.599,157.668
C07062=1038.811,172.118,400.151,170.172,40.599,157.668
C07063=1038.805,171.869,400.174,170.170,40.598,157.668
C07064=1038.800,171.620,400.197,170.167,40.598,157.667
C07065=1038.793,171.372,400.220,170.164,40.597,157.667
C07066=1038.786,171.122,400.243,170.162,40.597,157.667
C07067=1038.781,170.874,400.266,170.159,40.597,157.667
C07068=1038.775,170.625,400.289,170.157,40.596,157.667
C07069=1038.769,170.376,400.313,170.154,40.596,157.666
C07070=1038.763,170.128,400.336,170.151,40.596,157.666
C07071=1038.756,169.878,400.359,170.148,40.595,157.666
C07072=1038.750,169.629,400.382,170.146,40.594,157.666
C07073=1038.744,169.381,400.405,170.144,40.594,157.666
C07074=1038.739,169.132,400.428,170.141,40.593,157.665
C07075=1038.733,168.883,400.451,170.138,40.593,157.665
C07076=1038.727,168.634,400.474,170.135,40.593,157.665
C07077=1038.720,168.385,400.497,170.133,40.592,157.665
C07078=1038.714,168.136,400.520,170.131,40.592,157.665
C07079=1038.708,167.888,400.543,170.128,40.592,157.664
C07080=1038.703,167.639,400.566,170.125,40.591,157.664
C07081=1038.696,167.389,400.590,170.122,40.590,157.664
C07082=1038.690,167.141,400.612,170.120,40.590,157.664
C07083=1038.684,166.892,400.635,170.118,40.589,157.663
C07084=1038.678,166.643,400.658,170.115,40.589,157.663
C07085=1038.673,166.394,400.681,170.112,40.589,157.663
C07086=1038.667,166.145,400.704,170.110,40.588,157.663
C07087=1038.660,165.897,400.726,170.107,40.588,157.663
C07088=1038.654,165.648,400.750,170.105,40.588,157.662
C07089=1038.648,165.399,400.773,170.102,40.587,157.662
C07090=1038.642,165.150,400.796,170.099,40.587,157.662
C07091=1038.637,164.901,400.819,170.097,40.586,157.662
C07092=1038.630,164.652,400.841,170.094,40.586,157.662
C07093=1038.624,164.403,400.864,170.092,40.585,157.661
C07094=1038.619,164.155,400.887,170.090,40.585,157.661
C07095=1038.613,163.906,400.910,170.086,40.584,157.661
C07096=1038.607,163.657,400.933,170.084,40.584,157.661
C07097=1038.601,163.408,400.956,170.082,40.584,157.661
C07098=1038.595,163.159,400.978,170.079,40.583,157.660
C07099=1038.589,162.910,401.001,170.077,40.583,157.660
C07100=1038.584,162.662,401.024,170.075,40.582,157.660
C07101=1038.578,162.413,401.047,170.071,40.582,157.660
C07102=1038.572,162.163,401.069,170.069,40.581,157.659
C07103=1038.566,161.915,401.092,170.067,40.581,157.659
C07104=1038.560,161.666,401.115,170.064,40.580,157.659
C07105=1038.555,161.417,401.138,170.061,40.580,157.659
C07106=1038.548,161.168,401.160,170.059,40.579,157.659
C07107=1038.542,160.919,401.183,170.056,40.579,157.659
C07108=1038.536,160.670,401.206,170.054,40.579,157.658
C07109=1038.530,160.421,401.229,170.052,40.578,157.658
C07110=1038.525,160.172,401.252,170.049,40.578,157.658
C07111=1038.518,159.923,401.274,170.046,40.578,157.658
C07112=1038.512,159.674,401.296,170.044,40.577,157.658
C07113=1038.506,159.425,401.319,170.041,40.577,157.657
C07114=1038.500,159.177,401.342,170.039,40.576,157.657
C07115=1038.494,158.927,401.364,170.037,40.576,157.657
C07116=1038.488,158.678,401.386,170.034,40.576,157.657
C07117=1038.481,158.430,401.408,170.031,40.576,157.657
C07118=1038.476,158.180,401.431,170.029,40.576,157.657
C07119=1038.469,157.932,401.453,170.026,40.575,157.656
C07120=1038.463,157.683,401.475,170.024,40.575,157.656
C07121=1038.456,157.397,401.501,170.021,40.574,157.656
C07122=1038.449,157.113,401.526,170.019,40.574,157.656
C07123=1038.442,156.827,401.552,170.015,40.574,157.656
C07124=1038.436,156.542,401.578,170.012,40.573,157.655
C07125=1038.429,156.293,401.600,170.010,40.573,157.655
C07126=1038.423,156.045,401.622,170.008,40.573,157.655
C07127=1038.418,155.795,401.644,170.005,40.573,157.655
C07128=1038.411,155.547,401.667,170.003,40.573,157.655
C07129=1038.405,155.298,401.689,170.000,40.572,157.655
C07130=1038.399,155.048,401.711,169.997,40.572,157.654
C07131=1038.393,154.800,401.734,169.995,40.571,157.654
C07132=1038.387,154.551,401.755,169.993,40.571,157.654
C07133=1038.381,154.302,401.778,169.990,40.571,157.654
C07134=1038.375,154.053,401.800,169.988,40.571,157.654
C07135=1038.368,153.804,401.822,169.986,40.570,157.654
C07136=1038.362,153.555,401.844,169.982,40.570,157.653
C07137=1038.356,153.306,401.867,169.980,40.570,157.653
C07138=1038.350,153.057,401.888,169.978,40.570,157.653
C07139=1038.344,152.808,401.911,169.975,40.570,157.653
C07140=1038.337,152.559,401.932,169.973,40.569,157.653
C07141=1038.331,152.310,401.955,169.971,40.569,157.652
C07142=1038.326,152.061,401.977,169.969,40.569,157.652
C07143=1038.319,151.812,401.999,169.965,40.569,157.652
C07144=1038.313,151.563,402.021,169.963,40.568,157.652
C07145=1038.307,151.314,402.043,169.961,40.568,157.652
C07146=1038.301,151.066,402.065,169.958,40.568,157.652
C07147=1038.295,150.816,402.087,169.956,40.568,157.652
C07148=1038.289,150.568,402.109,169.954,40.567,157.651
C07149=1038.283,150.319,402.131,169.951,40.567,157.651
C07150=1038.277,150.069,402.152,169.948,40.567,157.651
C07151=1038.270,149.821,402.175,169.946,40.567,157.651
C07152=1038.265,149.571,402.197,169.944,40.566,157.651
C07153=1038.259,149.322,402.219,169.941,40.566,157.651
C07154=1038.252,149.073,402.241,169.939,40.566,157.650
C07155=1038.247,148.825,402.262,169.937,40.566,157.650
C07156=1038.240,148.576,402.284,169.935,40.565,157.650
C07157=1038.234,148.327,402.306,169.931,40.565,157.650
C07158=1038.228,148.078,402.328,169.929,40.565,157.650
C07159=1038.222,147.829,402.349,169.927,40.565,157.650
C07160=1038.215,147.580,402.372,169.924,40.565,157.650
C07161=1038.210,147.331,402.394,169.922,40.564,157.649
C07162=1038.204,147.081,402.416,169.920,40.564,157.649
C07163=1038.198,146.833,402.437,169.918,40.564,157.649
C07164=1038.192,146.584,402.459,169.914,40.564,157.649
C07165=1038.185,146.335,402.481,169.912,40.563,157.649
C07166=1038.179,146.086,402.503,169.910,40.563,157.649
C07167=1038.173,145.837,402.524,169.908,40.563,157.648
C07168=1038.166,145.588,402.545,169.905,40.563,157.648
C07169=1038.160,145.339,402.567,169.903,40.563,157.648
C07170=1038.154,145.090,402.588,169.901,40.563,157.648
C07171=1038.148,144.842,402.610,169.898,40.562,157.648
C07172=1038.142,144.592,402.632,169.896,40.562,157.648
C07173=1038.136,144.343,402.654,169.893,40.562,157.648
C07174=1038.129,144.094,402.675,169.891,40.562,157.648
C07175=1038.123,143.845,402.697,169.888,40.562,157.647
C07176=1038.118,143.596,402.718,169.886,40.562,157.647
C07177=1038.112,143.347,402.740,169.884,40.562,157.647
C07178=1038.105,143.098,402.762,169.882,40.561,157.647
C07179=1038.099,142.849,402.783,169.879,40.561,157.647
C07180=1038.093,142.599,402.805,169.877,40.561,157.647
C07181=1038.087,142.351,402.826,169.874,40.561,157.646
C07182=1038.081,142.102,402.847,169.872,40.560,157.646
C07183=1038.074,141.853,402.870,169.869,40.561,157.646
C07184=1038.068,141.604,402.891,169.867,40.560,157.646
C07185=1038.062,141.318,402.915,169.865,40.560,157.646
C07186=1038.055,141.033,402.940,169.862,40.560,157.646
C07187=1038.048,140.747,402.964,169.860,40.560,157.646
C07188=1038.041,140.462,402.989,169.856,40.559,157.645
C07189=1038.035,140.213,403.011,169.854,40.559,157.645
C07190=1038.029,139.964,403.033,169.852,40.559,157.645
C07191=1038.023,139.715,403.054,169.849,40.559,157.645
C07192=1038.016,139.466,403.075,169.847,40.558,157.645
C07193=1038.010,139.217,403.097,169.845,40.559,157.645
C07194=1038.004,138.968,403.118,169.843,40.558,157.644
C07195=1037.998,138.720,403.139,169.840,40.559,157.644
C07196=1037.992,138.470,403.161,169.837,40.558,157.644
C07197=1037.986,138.221,403.181,169.835,40.558,157.644
C07198=1037.979,137.972,403.203,169.833,40.558,157.644
C07199=1037.974,137.723,403.224,169.831,40.558,157.644
C07200=1037.968,137.474,403.246,169.828,40.558,157.644
C07201=1037.961,137.225,403.267,169.826,40.557,157.644
C07202=1037.955,136.976,403.289,169.824,40.558,157.644
C07203=1037.949,136.727,403.309,169.822,40.557,157.643
C07204=1037.942,136.478,403.330,169.819,40.557,157.643
C07205=1037.936,136.229,403.352,169.817,40.557,157.643
C07206=1037.931,135.980,403.373,169.814,40.557,157.643
C07207=1037.924,135.731,403.394,169.812,40.557,157.643
C07208=1037.918,135.481,403.415,169.810,40.557,157.643
C07209=1037.912,135.233,403.436,169.807,40.557,157.643
C07210=1037.905,134.984,403.457,169.805,40.556,157.642
C07211=1037.899,134.735,403.479,169.803,40.557,157.642
C07212=1037.894,134.486,403.500,169.801,40.556,157.642
C07213=1037.887,134.237,403.521,169.799,40.556,157.642
C07214=1037.881,133.987,403.542,169.796,40.556,157.642
C07215=1037.875,133.739,403.564,169.793,40.556,157.642
C07216=1037.869,133.489,403.584,169.791,40.556,157.642
C07217=1037.863,133.240,403.606,169.789,40.555,157.641
C07218=1037.857,132.992,403.627,169.787,40.556,157.641
C07219=1037.851,132.742,403.647,169.784,40.555,157.641
C07220=1037.844,132.493,403.669,169.782,40.556,157.641
C07221=1037.839,132.245,403.690,169.780,40.555,157.641
C07222=1037.832,131.995,403.710,169.778,40.555,157.641
C07223=1037.826,131.746,403.732,169.776,40.555,157.641
C07224=1037.820,131.498,403.753,169.773,40.555,157.641
C07225=1037.814,131.248,403.774,169.770,40.555,157.640
C07226=1037.808,130.999,403.795,169.768,40.554,157.640
C07227=1037.802,130.750,403.815,169.766,40.555,157.640
C07228=1037.796,130.501,403.837,169.764,40.554,157.640
C07229=1037.790,130.252,403.857,169.762,40.554,157.640
C07230=1037.783,130.003,403.878,169.759,40.555,157.640
C07231=1037.777,129.753,403.899,169.757,40.554,157.640
C07232=1037.771,129.505,403.919,169.755,40.555,157.640
C07233=1037.764,129.255,403.940,169.753,40.554,157.640
C07234=1037.758,129.006,403.961,169.750,40.554,157.639
C07235=1037.752,128.757,403.981,169.748,40.555,157.639
C07236=1037.745,128.508,404.002,169.745,40.554,157.639
C07237=1037.740,128.259,404.023,169.743,40.554,157.639
C07238=1037.733,128.010,404.044,169.741,40.554,157.639
C07239=1037.726,127.761,404.064,169.738,40.554,157.639
C07240=1037.721,127.512,404.086,169.736,40.555,157.639
C07241=1037.714,127.263,404.106,169.734,40.554,157.639
C07242=1037.708,127.015,404.127,169.732,40.554,157.639
C07243=1037.701,126.765,404.147,169.730,40.554,157.638
C07244=1037.695,126.515,404.168,169.728,40.554,157.638
C07245=1037.689,126.267,404.188,169.725,40.554,157.638
C07246=1037.682,126.018,404.209,169.722,40.554,157.638
C07247=1037.677,125.769,404.230,169.720,40.554,157.638
C07248=1037.670,125.520,404.250,169.718,40.554,157.638
C07249=1037.663,125.234,404.274,169.715,40.554,157.638
C07250=1037.656,124.949,404.298,169.713,40.554,157.638
C07251=1037.649,124.662,404.321,169.710,40.554,157.638
C07252=1037.642,124.377,404.345,169.708,40.554,157.637
C07253=1037.635,124.127,404.365,169.706,40.554,157.637
C07254=1037.630,123.879,404.386,169.704,40.554,157.637
C07255=1037.623,123.629,404.407,169.701,40.554,157.637
C07256=1037.617,123.380,404.427,169.699,40.554,157.637
C07257=1037.611,123.131,404.448,169.696,40.554,157.637
C07258=1037.605,122.882,404.468,169.694,40.554,157.637
C07259=1037.598,122.633,404.488,169.692,40.554,157.637
C07260=1037.592,122.385,404.509,169.690,40.554,157.637
C07261=1037.586,122.135,404.530,169.687,40.554,157.636
C07262=1037.580,121.886,404.550,169.685,40.553,157.636
C07263=1037.574,121.636,404.570,169.683,40.554,157.636
C07264=1037.568,121.388,404.592,169.681,40.553,157.636
C07265=1037.561,121.138,404.612,169.679,40.553,157.636
C07266=1037.555,120.890,404.632,169.677,40.554,157.636
C07267=1037.550,120.641,404.652,169.675,40.553,157.636
C07268=1037.544,120.391,404.673,169.672,40.554,157.636
C07269=1037.537,120.143,404.693,169.669,40.553,157.635
C07270=1037.531,119.893,404.714,169.667,40.553,157.635
C07271=1037.525,119.644,404.734,169.665,40.553,157.635
C07272=1037.519,119.395,404.755,169.663,40.553,157.635
C07273=1037.513,119.146,404.775,169.661,40.553,157.635
C07274=1037.506,118.897,404.796,169.659,40.553,157.635
C07275=1037.501,118.648,404.816,169.657,40.553,157.635
